{attribute 'no_assign'}
{attribute 'no_explicit_call' := 'do not call this function block directly'}
FUNCTION_BLOCK ListAppendGenericTest EXTENDS TOF_Testing.SingleCycleTest
VAR_STAT
	{attribute 'hide'}
	_ClassName : STRING := __POUNAME();
END_VAR
VAR
	_List : TOF_Collections.IList;
	_Values : ARRAY [0..5] OF STRING := ['String0', 'String1', 'String2', 'String3', 'String4', 'String5'];
END_VAR

(*!
<summary>Clears the fixture before the runner publishes the result.</summary>
<description>
Also runs after an unexpected exception interrupts the case.
</description>
*)
METHOD PROTECTED AfterTest
_List.Clear();
END_METHOD

//! <summary>Borrows the concrete class name. Callers must not modify it.</summary>
{attribute 'monitoring' := 'call'}
PROPERTY ClassName : REFERENCE TO STRING
GET
ClassName REF= _ClassName;
END_GET
END_PROPERTY

(*!
<summary>Checks appending borrowed strings without cloning or adopting them.</summary>
*)
METHOD PROTECTED ExecuteTest
VAR
	entry : TOF_Core.GENERIC_VALUE;
	expected : ARRAY [0..2] OF STRING := ['String0', 'String1', 'String2'];
	i : DINT;
END_VAR
entry := TOF_Core.GenericValueFactory.FromStringReference(value := _Values[0]);
_List.AppendGeneric(value := entry);

entry := TOF_Core.GenericValueFactory.FromStringReference(value := _Values[1]);
_List.AppendGeneric(value := entry);

entry := TOF_Core.GenericValueFactory.FromStringReference(value := _Values[2]);
_List.AppendGeneric(value := entry);

Assert.ThatBool(
	actual := _List.Get(index := 2).Address = entry.Address AND_THEN NOT _List.Get(index := 2).IsMemoryOwner,
	message := "AppendGeneric must retain the borrowed address and ownership mode"
).IsTrue();

Assert.ThatDInt(
	actual := _List.Length,
	message := "Unexpected sequence after AppendGeneric length"
).ToBe(expected := DINT#3);

FOR i := 0 TO 2 DO
	Assert.ThatString(
		actual := _List.Get(index := i).AsString255(),
		message := TOF_Core.WideStrings.Concat255("Unexpected sequence after AppendGeneric at index ", TO_WSTRING(i))
	).ToBe(expected := expected[i]);
END_FOR
END_METHOD

(*!
<summary>Binds the list fixture for this case.</summary>
<description>
Stores a borrowed interface without invoking the fixture. The owning group keeps it alive and
reserves it for this case. TestElement initializes the name and parent.
</description>
<param name="name">Display name of this case.</param>
<param name="parent">Group that owns this case.</param>
<param name="list">Required live list reserved for this case.</param>
*)
METHOD FB_init : BOOL
VAR_INPUT
	bInitRetains: BOOL; // TRUE: the retain variables are initialized (reset warm / reset cold)
	bInCopyCode: BOOL; // TRUE: the instance will be copied to the copy code afterward (online change)
	name : WSTRING;
	parent : TOF_Testing.ITestElement;
	list : TOF_Collections.IList;
END_VAR
_List := list;
FB_init := TRUE;
END_METHOD

//! <summary>Borrows the compiler-initialized namespace name. Callers must not modify it.</summary>
{attribute 'monitoring' := 'call'}
PROPERTY NamespaceName : REFERENCE TO STRING
GET
NamespaceName REF= CurrentNamespace.Name;
END_GET
END_PROPERTY

//! <summary>Reports the concrete instance size in bytes.</summary>
{attribute 'monitoring' := 'call'}
PROPERTY SelfSize : ULINT
GET
SelfSize := XSIZEOF(THIS^);
END_GET
END_PROPERTY

END_FUNCTION_BLOCK

// ---- Tests/Collections/ListInsertGenericTest.TcPOU
(*
SPDX-FileCopyrightText: c 2026 Oleksandr Tiutyk <trofimich@gmail.com>
SPDX-License-Identifier: MIT
License: https://opensource.org/license/mit
*)

(*!
<summary>Checks borrowed insertion and suffix order.</summary>
<description>
Borrows a group-owned list reserved for this case. Use from one task at a stable address.
Teardown clears the list before publication.
</description>
*)

{attribute 'no_assign'}
{attribute 'no_explicit_call' := 'do not call this function block directly'}
FUNCTION_BLOCK ListInsertGenericTest EXTENDS TOF_Testing.SingleCycleTest
VAR_STAT
	{attribute 'hide'}
	_ClassName : STRING := __POUNAME();
END_VAR
VAR
	_List : TOF_Collections.IList;
	_Values : ARRAY [0..5] OF STRING := ['String0', 'String1', 'String2', 'String3', 'String4', 'String5'];
END_VAR

(*!
<summary>Clears the fixture before the runner publishes the result.</summary>
<description>
Also runs after an unexpected exception interrupts the case.
</description>
*)
METHOD PROTECTED AfterTest
_List.Clear();
END_METHOD

//! <summary>Borrows the concrete class name. Callers must not modify it.</summary>
{attribute 'monitoring' := 'call'}
PROPERTY ClassName : REFERENCE TO STRING
GET
ClassName REF= _ClassName;
END_GET
END_PROPERTY

(*!
<summary>Checks borrowed insertion and suffix order.</summary>
*)
METHOD PROTECTED ExecuteTest
VAR
	values : ARRAY [0..5] OF STRING := ['String0', 'String1', 'String2', 'String3', 'String4', 'String5'];
	entry : TOF_Core.GENERIC_VALUE;
	expected : ARRAY [0..3] OF STRING := ['String0', 'String5', 'String1', 'String2'];
	i : DINT;
END_VAR
_List.AppendCopy(value := values[0]);
_List.AppendCopy(value := values[1]);
_List.AppendCopy(value := values[2]);

entry := TOF_Core.GenericValueFactory.FromStringReference(value := _Values[5]);
_List.InsertGeneric(index := 1, value := entry);

Assert.ThatBool(
	actual := _List.Get(index := 1).Address = entry.Address AND_THEN NOT _List.Get(index := 1).IsMemoryOwner,
	message := "InsertGeneric must retain the borrowed address and ownership mode"
).IsTrue();

Assert.ThatDInt(
	actual := _List.Length,
	message := "Unexpected sequence after InsertGeneric length"
).ToBe(expected := DINT#4);

FOR i := 0 TO 3 DO
	Assert.ThatString(
		actual := _List.Get(index := i).AsString255(),
		message := TOF_Core.WideStrings.Concat255("Unexpected sequence after InsertGeneric at index ", TO_WSTRING(i))
	).ToBe(expected := expected[i]);
END_FOR
END_METHOD

(*!
<summary>Binds the list fixture for this case.</summary>
<description>
Stores a borrowed interface without invoking the fixture. The owning group keeps it alive and
reserves it for this case. TestElement initializes the name and parent.
</description>
<param name="name">Display name of this case.</param>
<param name="parent">Group that owns this case.</param>
<param name="list">Required live list reserved for this case.</param>
*)
METHOD FB_init : BOOL
VAR_INPUT
	bInitRetains: BOOL; // TRUE: the retain variables are initialized (reset warm / reset cold)
	bInCopyCode: BOOL; // TRUE: the instance will be copied to the copy code afterward (online change)
	name : WSTRING;
	parent : TOF_Testing.ITestElement;
	list : TOF_Collections.IList;
END_VAR
_List := list;
FB_init := TRUE;
END_METHOD

//! <summary>Borrows the compiler-initialized namespace name. Callers must not modify it.</summary>
{attribute 'monitoring' := 'call'}
PROPERTY NamespaceName : REFERENCE TO STRING
GET
NamespaceName REF= CurrentNamespace.Name;
END_GET
END_PROPERTY

//! <summary>Reports the concrete instance size in bytes.</summary>
{attribute 'monitoring' := 'call'}
PROPERTY SelfSize : ULINT
GET
SelfSize := XSIZEOF(THIS^);
END_GET
END_PROPERTY

END_FUNCTION_BLOCK

// ---- Tests/Collections/ListGetAndSetGenericTest.TcPOU
(*
SPDX-FileCopyrightText: c 2026 Oleksandr Tiutyk <trofimich@gmail.com>
SPDX-License-Identifier: MIT
License: https://opensource.org/license/mit
*)

(*!
<summary>Checks borrowed replacement and the surrounding entries.</summary>
<description>
Borrows a group-owned list reserved for this case. Use from one task at a stable address.
Teardown clears the list before publication.
</description>
*)

{attribute 'no_assign'}
{attribute 'no_explicit_call' := 'do not call this function block directly'}
FUNCTION_BLOCK ListGetAndSetGenericTest EXTENDS TOF_Testing.SingleCycleTest
VAR_STAT
	{attribute 'hide'}
	_ClassName : STRING := __POUNAME();
END_VAR
VAR
	_List : TOF_Collections.IList;
	_Values : ARRAY [0..5] OF STRING := ['String0', 'String1', 'String2', 'String3', 'String4', 'String5'];
END_VAR

(*!
<summary>Clears the fixture before the runner publishes the result.</summary>
<description>
Also runs after an unexpected exception interrupts the case.
</description>
*)
METHOD PROTECTED AfterTest
_List.Clear();
END_METHOD

//! <summary>Borrows the concrete class name. Callers must not modify it.</summary>
{attribute 'monitoring' := 'call'}
PROPERTY ClassName : REFERENCE TO STRING
GET
ClassName REF= _ClassName;
END_GET
END_PROPERTY

(*!
<summary>Checks borrowed replacement and the surrounding entries.</summary>
*)
METHOD PROTECTED ExecuteTest
VAR
	values : ARRAY [0..5] OF STRING := ['String0', 'String1', 'String2', 'String3', 'String4', 'String5'];
	entry : TOF_Core.GENERIC_VALUE;
	expected : ARRAY [0..2] OF STRING := ['String0', 'String4', 'String2'];
	i : DINT;
END_VAR
_List.AppendCopy(value := values[0]);
_List.AppendCopy(value := values[1]);
_List.AppendCopy(value := values[2]);

entry := TOF_Core.GenericValueFactory.FromStringReference(value := _Values[4]);
_List.SetGeneric(index := 1, value := entry);

Assert.ThatBool(
	actual := _List.Get(index := 1).Address = entry.Address AND_THEN NOT _List.Get(index := 1).IsMemoryOwner,
	message := "SetGeneric must retain the borrowed address and ownership mode"
).IsTrue();

Assert.ThatDInt(
	actual := _List.Length,
	message := "Unexpected sequence after GetAndSetGeneric length"
).ToBe(expected := DINT#3);

FOR i := 0 TO 2 DO
	Assert.ThatString(
		actual := _List.Get(index := i).AsString255(),
		message := TOF_Core.WideStrings.Concat255("Unexpected sequence after GetAndSetGeneric at index ", TO_WSTRING(i))
	).ToBe(expected := expected[i]);
END_FOR
END_METHOD

(*!
<summary>Binds the list fixture for this case.</summary>
<description>
Stores a borrowed interface without invoking the fixture. The owning group keeps it alive and
reserves it for this case. TestElement initializes the name and parent.
</description>
<param name="name">Display name of this case.</param>
<param name="parent">Group that owns this case.</param>
<param name="list">Required live list reserved for this case.</param>
*)
METHOD FB_init : BOOL
VAR_INPUT
	bInitRetains: BOOL; // TRUE: the retain variables are initialized (reset warm / reset cold)
	bInCopyCode: BOOL; // TRUE: the instance will be copied to the copy code afterward (online change)
	name : WSTRING;
	parent : TOF_Testing.ITestElement;
	list : TOF_Collections.IList;
END_VAR
_List := list;
FB_init := TRUE;
END_METHOD

//! <summary>Borrows the compiler-initialized namespace name. Callers must not modify it.</summary>
{attribute 'monitoring' := 'call'}
PROPERTY NamespaceName : REFERENCE TO STRING
GET
NamespaceName REF= CurrentNamespace.Name;
END_GET
END_PROPERTY

//! <summary>Reports the concrete instance size in bytes.</summary>
{attribute 'monitoring' := 'call'}
PROPERTY SelfSize : ULINT
GET
SelfSize := XSIZEOF(THIS^);
END_GET
END_PROPERTY

END_FUNCTION_BLOCK

// ---- Tests/Collections/Dynamic/DynamicListClearTest.TcPOU
(*
SPDX-FileCopyrightText: c 2026 Oleksandr Tiutyk <trofimich@gmail.com>
SPDX-License-Identifier: MIT
License: https://opensource.org/license/mit
*)

(*!
<summary>Checks release of populated storage and fresh allocation on reuse.</summary>
<description>
Owns a list and its copied entries. Use from one task at a stable address.
Teardown clears surviving entries before publication.
</description>
*)

{attribute 'no_assign'}
{attribute 'no_explicit_call' := 'do not call this function block directly'}
FUNCTION_BLOCK DynamicListClearTest EXTENDS TOF_Testing.SingleCycleTest
VAR_STAT
	{attribute 'hide'}
	_ClassName : STRING := __POUNAME();
END_VAR
VAR
	_List : TOF_Collections.List<0>(valueValidator := 0);
END_VAR

(*!
<summary>Checks release of populated storage and fresh allocation on reuse.</summary>
*)
METHOD PROTECTED ExecuteTest
VAR
	values : ARRAY [0..5] OF STRING := ['String0', 'String1', 'String2', 'String3', 'String4', 'String5'];
END_VAR
_List.AppendCopy(value := values[0]);
_List.AppendCopy(value := values[1]);
_List.AppendCopy(value := values[2]);
_List.AppendCopy(value := values[3]);
_List.AppendCopy(value := values[4]);
_List.AppendCopy(value := values[5]);

Assert.ThatBool(
	actual := _List.Length = 6 AND_THEN _List.Capacity >= 6,
	message := "Clear fixture must contain six live entries"
).IsTrue();

_List.Clear();

Assert.ThatBool(
	actual := _List.Empty AND_THEN _List.Length = 0 AND_THEN _List.Capacity = 0,
	message := "Clear must empty the dynamic list and release its capacity"
).IsTrue();

_List.AppendCopy(value := values[5]);

Assert.ThatBool(
	actual := _List.Length = 1 AND_THEN _List.Get(index := 0).AsString255() = 'String5',
	message := "The cleared list must accept a fresh value"
).IsTrue();
END_METHOD

(*!
<summary>Clears the fixture before the runner publishes the result.</summary>
<description>
Also runs after an unexpected exception interrupts the case.
</description>
*)
METHOD PROTECTED AfterTest
_List.Clear();
END_METHOD

//! <summary>Borrows the concrete class name. Callers must not modify it.</summary>
{attribute 'monitoring' := 'call'}
PROPERTY ClassName : REFERENCE TO STRING
GET
ClassName REF= _ClassName;
END_GET
END_PROPERTY

//! <summary>Borrows the compiler-initialized namespace name. Callers must not modify it.</summary>
{attribute 'monitoring' := 'call'}
PROPERTY NamespaceName : REFERENCE TO STRING
GET
NamespaceName REF= CurrentNamespace.Name;
END_GET
END_PROPERTY

//! <summary>Reports the concrete instance size in bytes.</summary>
{attribute 'monitoring' := 'call'}
PROPERTY SelfSize : ULINT
GET
SelfSize := XSIZEOF(THIS^);
END_GET
END_PROPERTY

END_FUNCTION_BLOCK

// ---- Tests/Collections/Static/StaticListTestGroup.TcPOU
(*
SPDX-FileCopyrightText: c 2026 Oleksandr Tiutyk <trofimich@gmail.com>
SPDX-License-Identifier: MIT
License: https://opensource.org/license/mit
*)

(*!
<summary>Groups fixed-capacity list copying, borrowing, editing, search, sorting and overflow cases.</summary>
<description>
Owns the cases, their fixed registration array and any fixtures borrowed by the cases.
Each borrowed fixture is reserved for its case throughout the group lifetime. Use from one task at a stable address.
</description>
*)

{attribute 'no_assign'}
{attribute 'no_explicit_call' := 'do not call this function block directly'}
FUNCTION_BLOCK StaticListTestGroup EXTENDS TOF_Testing.TestGroup<16>
VAR_STAT
	{attribute 'hide'}
	_ClassName : STRING := __POUNAME();
END_VAR
VAR
	_AppendList : TOF_Collections.List<8>(valueValidator := 0);
	_InsertList : TOF_Collections.List<8>(valueValidator := 0);
	_GetAndSetList : TOF_Collections.List<8>(valueValidator := 0);
	_FindList : TOF_Collections.List<8>(valueValidator := 0);
	_ContainsList : TOF_Collections.List<8>(valueValidator := 0);
	_ContainsGenericList : TOF_Collections.List<8>(valueValidator := 0);
	_RemoveFirstList : TOF_Collections.List<8>(valueValidator := 0);
	_RemoveMatchedList : TOF_Collections.List<8>(valueValidator := 0);
	_RemoveAtList : TOF_Collections.List<8>(valueValidator := 0);
	_SwapList : TOF_Collections.List<8>(valueValidator := 0);
	_AppendGenericList : TOF_Collections.List<8>(valueValidator := 0);
	_InsertGenericList : TOF_Collections.List<8>(valueValidator := 0);
	_GetAndSetGenericList : TOF_Collections.List<8>(valueValidator := 0);

	_Append : ListAppendTest(name := "Append", parent := THIS^, list := _AppendList);
	_Insert : ListInsertTest(name := "Insert", parent := THIS^, list := _InsertList);
	_GetAndSet : ListGetAndSetTest(name := "GetAndSet", parent := THIS^, list := _GetAndSetList);
	_Find : ListFindTest(name := "Find", parent := THIS^, list := _FindList);
	_Contains : ListContainsTest(name := "Contains", parent := THIS^, list := _ContainsList);
	_ContainsGeneric : ListContainsGenericTest(name := "ContainsGeneric", parent := THIS^, list := _ContainsGenericList);
	_RemoveFirst : ListRemoveFirstTest(name := "RemoveFirst", parent := THIS^, list := _RemoveFirstList);
	_RemoveMatched : ListRemoveMatchedTest(name := "RemoveMatched", parent := THIS^, list := _RemoveMatchedList);
	_RemoveAt : ListRemoveAtTest(name := "RemoveAt", parent := THIS^, list := _RemoveAtList);
	_Swap : ListSwapTest(name := "Swap", parent := THIS^, list := _SwapList);
	_Sort : StaticListSortTest(name := "Sort", parent := THIS^);
	_AppendGeneric : ListAppendGenericTest(name := "AppendGeneric", parent := THIS^, list := _AppendGenericList);
	_InsertGeneric : ListInsertGenericTest(name := "InsertGeneric", parent := THIS^, list := _InsertGenericList);
	_GetAndSetGeneric : ListGetAndSetGenericTest(
		name := "GetAndSetGeneric",
		parent := THIS^,
		list := _GetAndSetGenericList
	);
	_Clear : StaticListClearTest(name := "Clear", parent := THIS^);
	_Overflow : StaticListOverflowTest(name := "Overflow", parent := THIS^);

	_Children : ARRAY [0.._ChildCount - 1] OF TOF_Testing.ITestElement :=
	[
		_Append,
		_Insert,
		_GetAndSet,
		_Find,
		_Contains,
		_ContainsGeneric,
		_RemoveFirst,
		_RemoveMatched,
		_RemoveAt,
		_Swap,
		_Sort,
		_AppendGeneric,
		_InsertGeneric,
		_GetAndSetGeneric,
		_Clear,
		_Overflow
	];
END_VAR

//! <summary>Borrows the fixed child array. Callers must not modify it.</summary>
{attribute 'monitoring' := 'call'}
PROPERTY Children : REFERENCE TO ARRAY [0.._ChildCount - 1] OF TOF_Testing.ITestElement
GET
Children REF= _Children;
END_GET
END_PROPERTY

//! <summary>Borrows the concrete class name. Callers must not modify it.</summary>
{attribute 'monitoring' := 'call'}
PROPERTY ClassName : REFERENCE TO STRING
GET
ClassName REF= _ClassName;
END_GET
END_PROPERTY

//! <summary>Borrows the compiler-initialized namespace name. Callers must not modify it.</summary>
{attribute 'monitoring' := 'call'}
PROPERTY NamespaceName : REFERENCE TO STRING
GET
NamespaceName REF= CurrentNamespace.Name;
END_GET
END_PROPERTY

//! <summary>Reports the concrete instance size in bytes.</summary>
{attribute 'monitoring' := 'call'}
PROPERTY SelfSize : ULINT
GET
SelfSize := XSIZEOF(THIS^);
END_GET
END_PROPERTY

END_FUNCTION_BLOCK

// ---- Tests/Collections/Static/StaticListSortTest.TcPOU
(*
SPDX-FileCopyrightText: c 2026 Oleksandr Tiutyk <trofimich@gmail.com>
SPDX-License-Identifier: MIT
License: https://opensource.org/license/mit
*)

(*!
<summary>Checks ascending sorting of a full list with duplicate strings and reverse lookup.</summary>
<description>
Owns a list and its copied entries. Use from one task at a stable address.
Teardown clears surviving entries before publication.
</description>
*)

{attribute 'no_assign'}
{attribute 'no_explicit_call' := 'do not call this function block directly'}
FUNCTION_BLOCK StaticListSortTest EXTENDS TOF_Testing.SingleCycleTest
VAR_STAT
	{attribute 'hide'}
	_ClassName : STRING := __POUNAME();
END_VAR
VAR
	_List : TOF_Collections.List<8>(valueValidator := 0);
	_Predicate : ListStringPredicate;
END_VAR

(*!
<summary>Checks ascending sorting of a full list with duplicate strings and reverse lookup.</summary>
*)
METHOD PROTECTED ExecuteTest
VAR
	values : ARRAY [0..5] OF STRING := ['String0', 'String1', 'String2', 'String3', 'String4', 'String5'];
	expected : ARRAY [0..7] OF STRING :=
		['String0', 'String1', 'String2', 'String2', 'String2', 'String3', 'String4', 'String5'];
	i : DINT;
	index : TOF_Core.DINT_INDEX;
	found : BOOL;
	entry : TOF_Core.GENERIC_VALUE;
END_VAR
_List.AppendCopy(value := values[5]);
_List.AppendCopy(value := values[4]);
_List.AppendCopy(value := values[3]);
_List.AppendCopy(value := values[2]);
_List.AppendCopy(value := values[2]);
_List.AppendCopy(value := values[2]);
_List.AppendCopy(value := values[1]);
_List.AppendCopy(value := values[0]);

_List.Sort(comparer := TOF_Comparison.StandardComparers.StringComparer);

Assert.ThatDInt(
	actual := _List.Length,
	message := "Ascending sort length"
).ToBe(expected := DINT#8);

FOR i := 0 TO 7 DO
	Assert.ThatString(
		actual := _List.Get(index := i).AsString255(),
		message := TOF_Core.WideStrings.Concat255("Ascending sort at index ", TO_WSTRING(i))
	).ToBe(expected := expected[i]);
END_FOR

_Predicate.Expected := 'String3';

found := _List.FindSingle(
	predicate := _Predicate,
	searchDirection := TOF_Core.SEARCH_DIRECTION.FROM_END,
	value => entry,
	index => index
);

Assert.ThatBool(
	actual := found AND_THEN index = 5 AND_THEN entry.AsString255() = 'String3',
	message := "Reverse lookup must return String3 at its current position after sorting"
).IsTrue();
END_METHOD

(*!
<summary>Clears the fixture before the runner publishes the result.</summary>
<description>
Also runs after an unexpected exception interrupts the case.
</description>
*)
METHOD PROTECTED AfterTest
_List.Clear();
END_METHOD

//! <summary>Borrows the concrete class name. Callers must not modify it.</summary>
{attribute 'monitoring' := 'call'}
PROPERTY ClassName : REFERENCE TO STRING
GET
ClassName REF= _ClassName;
END_GET
END_PROPERTY

//! <summary>Borrows the compiler-initialized namespace name. Callers must not modify it.</summary>
{attribute 'monitoring' := 'call'}
PROPERTY NamespaceName : REFERENCE TO STRING
GET
NamespaceName REF= CurrentNamespace.Name;
END_GET
END_PROPERTY

//! <summary>Reports the concrete instance size in bytes.</summary>
{attribute 'monitoring' := 'call'}
PROPERTY SelfSize : ULINT
GET
SelfSize := XSIZEOF(THIS^);
END_GET
END_PROPERTY

END_FUNCTION_BLOCK

// ---- Tests/Collections/Static/StaticListClearTest.TcPOU
(*
SPDX-FileCopyrightText: c 2026 Oleksandr Tiutyk <trofimich@gmail.com>
SPDX-License-Identifier: MIT
License: https://opensource.org/license/mit
*)

(*!
<summary>Checks clearing a full inline list and reusing all eight slots.</summary>
<description>
Owns a list and its copied entries. Use from one task at a stable address.
Teardown clears surviving entries before publication.
</description>
*)

{attribute 'no_assign'}
{attribute 'no_explicit_call' := 'do not call this function block directly'}
FUNCTION_BLOCK StaticListClearTest EXTENDS TOF_Testing.SingleCycleTest
VAR_STAT
	{attribute 'hide'}
	_ClassName : STRING := __POUNAME();
END_VAR
VAR
	_List : TOF_Collections.List<8>(valueValidator := 0);
END_VAR

(*!
<summary>Checks clearing a full inline list and reusing all eight slots.</summary>
*)
METHOD PROTECTED ExecuteTest
VAR
	values : ARRAY [0..5] OF STRING := ['String0', 'String1', 'String2', 'String3', 'String4', 'String5'];
END_VAR
_List.AppendCopy(value := values[0]);
_List.AppendCopy(value := values[1]);
_List.AppendCopy(value := values[2]);
_List.AppendCopy(value := values[3]);
_List.AppendCopy(value := values[4]);
_List.AppendCopy(value := values[5]);
_List.AppendCopy(value := values[0]);
_List.AppendCopy(value := values[1]);

Assert.ThatBool(
	actual := _List.Full,
	message := "Clear fixture must start full"
).IsTrue();

_List.Clear();

Assert.ThatBool(
	actual := _List.Empty AND_THEN _List.Length = 0 AND_THEN _List.Capacity = 8 AND_THEN NOT _List.Full,
	message := "Clear must empty the list while retaining its inline capacity"
).IsTrue();

_List.AppendCopy(value := values[5]);
_List.AppendCopy(value := values[4]);
_List.AppendCopy(value := values[3]);
_List.AppendCopy(value := values[2]);
_List.AppendCopy(value := values[1]);
_List.AppendCopy(value := values[0]);
_List.AppendCopy(value := values[3]);
_List.AppendCopy(value := values[4]);

Assert.ThatBool(
	actual := _List.Full AND_THEN _List.Get(index := 0).AsString255() = 'String5'
		AND_THEN _List.Get(index := 7).AsString255() = 'String4',
	message := "Refill must occupy all slots with the new head and tail"
).IsTrue();
END_METHOD

(*!
<summary>Clears the fixture before the runner publishes the result.</summary>
<description>
Also runs after an unexpected exception interrupts the case.
</description>
*)
METHOD PROTECTED AfterTest
_List.Clear();
END_METHOD

//! <summary>Borrows the concrete class name. Callers must not modify it.</summary>
{attribute 'monitoring' := 'call'}
PROPERTY ClassName : REFERENCE TO STRING
GET
ClassName REF= _ClassName;
END_GET
END_PROPERTY

//! <summary>Borrows the compiler-initialized namespace name. Callers must not modify it.</summary>
{attribute 'monitoring' := 'call'}
PROPERTY NamespaceName : REFERENCE TO STRING
GET
NamespaceName REF= CurrentNamespace.Name;
END_GET
END_PROPERTY

//! <summary>Reports the concrete instance size in bytes.</summary>
{attribute 'monitoring' := 'call'}
PROPERTY SelfSize : ULINT
GET
SelfSize := XSIZEOF(THIS^);
END_GET
END_PROPERTY

END_FUNCTION_BLOCK

// ---- Tests/Collections/Static/StaticListOverflowTest.TcPOU
(*
SPDX-FileCopyrightText: c 2026 Oleksandr Tiutyk <trofimich@gmail.com>
SPDX-License-Identifier: MIT
License: https://opensource.org/license/mit
*)

(*!
<summary>Checks overflow at eight elements and reuse after freeing a slot.</summary>
<description>
Owns a list and its copied entries. Use from one task at a stable address.
Teardown clears surviving entries before publication.
</description>
*)

{attribute 'no_assign'}
{attribute 'no_explicit_call' := 'do not call this function block directly'}
FUNCTION_BLOCK StaticListOverflowTest EXTENDS TOF_Testing.SingleCycleTest
VAR_STAT
	{attribute 'hide'}
	_ClassName : STRING := __POUNAME();
END_VAR
VAR
	_List : TOF_Collections.List<8>(valueValidator := 0);
END_VAR

(*!
<summary>Checks overflow at eight elements and reuse after freeing a slot.</summary>
*)
METHOD PROTECTED ExecuteTest
VAR
	values : ARRAY [1..9] OF INT := [1, 2, 3, 4, 5, 6, 7, 8, 9];
	i : DINT;

	exceptionCode : __SYSTEM.ExceptionCode;
	caught : TOF_Core.IException;
	fullException : TOF_Core.IStaticCollectionFullException;
END_VAR
FOR i := 1 TO 8 DO
	_List.AppendCopy(value := values[i]);
END_FOR

Assert.ThatBool(
	actual := _List.Full,
	message := "Overflow fixture must start full"
).IsTrue();

__TRY
	_List.AppendCopy(value := values[9]);
__CATCH(exceptionCode)
	caught := TOF_Core.ExceptionManager.GetLastException(
		exceptionCode := exceptionCode,
		catchPointNamespaceName := NamespaceName,
		catchPointPOUName := __POUNAME(),
		catchPointPosition := __POSITION()
	);
__ENDTRY

Assert.ThatBool(
	actual := __QUERYINTERFACE(caught, fullException),
	message := "Appending beyond capacity must raise StaticCollectionFullException"
).IsTrue();

Assert.ThatBool(
	actual := _List.Full AND_THEN _List.Length = 8 AND_THEN _List.Capacity = 8,
	message := "Rejected append must preserve length and capacity"
).IsTrue();

FOR i := 1 TO 8 DO
	Assert.ThatInt(
		actual := _List.Get(index := i - 1).AsInt(),
		message := TOF_Core.WideStrings.Concat255("Overflow must preserve member ", TO_WSTRING(i))
	).ToBe(expected := values[i]);
END_FOR

_List.RemoveAt(index := 7);
_List.AppendCopy(value := values[9]);

Assert.ThatBool(
	actual := _List.Full AND_THEN _List.Get(index := 7).AsInt() = INT#9,
	message := "Appending after removal must reuse the freed slot"
).IsTrue();
END_METHOD

(*!
<summary>Clears the fixture before the runner publishes the result.</summary>
<description>
Also runs after an unexpected exception interrupts the case.
</description>
*)
METHOD PROTECTED AfterTest
_List.Clear();
END_METHOD

//! <summary>Borrows the concrete class name. Callers must not modify it.</summary>
{attribute 'monitoring' := 'call'}
PROPERTY ClassName : REFERENCE TO STRING
GET
ClassName REF= _ClassName;
END_GET
END_PROPERTY

//! <summary>Borrows the compiler-initialized namespace name. Callers must not modify it.</summary>
{attribute 'monitoring' := 'call'}
PROPERTY NamespaceName : REFERENCE TO STRING
GET
NamespaceName REF= CurrentNamespace.Name;
END_GET
END_PROPERTY

//! <summary>Reports the concrete instance size in bytes.</summary>
{attribute 'monitoring' := 'call'}
PROPERTY SelfSize : ULINT
GET
SelfSize := XSIZEOF(THIS^);
END_GET
END_PROPERTY

END_FUNCTION_BLOCK

// ---- Tests/Collections/Dynamic/DynamicStackTestGroup.TcPOU
(*
SPDX-FileCopyrightText: c 2026 Oleksandr Tiutyk <trofimich@gmail.com>
SPDX-License-Identifier: MIT
License: https://opensource.org/license/mit
*)

(*!
<summary>Groups dynamic stack storage, LIFO order, cursors and ownership cases.</summary>
<description>
Owns the cases, their fixed registration array and any fixtures borrowed by the cases.
Each borrowed fixture is reserved for its case throughout the group lifetime. Use from one task at a stable address.
</description>
*)

{attribute 'no_assign'}
{attribute 'no_explicit_call' := 'do not call this function block directly'}
FUNCTION_BLOCK DynamicStackTestGroup EXTENDS TOF_Testing.TestGroup<11>
VAR_STAT
	{attribute 'hide'}
	_ClassName : STRING := __POUNAME();
END_VAR
VAR
	_Validator : TOF_Core.GenericValueTypeValidator(typeClass := TOF_Core.GENERIC_TYPE_CLASS.INT_16);
	_OwnedObjectCleanupStack : TOF_Collections.Stack<0>(valueValidator := 0);
	_ValidatorRejectionStack : TOF_Collections.Stack<0>(valueValidator := _Validator);
	_IndexedAccessAndEnumerationStack : TOF_Collections.Stack<0>(valueValidator := 0);
	_EmptyAndIndexBoundsStack : TOF_Collections.Stack<0>(valueValidator := 0);
	_CopiedAndBorrowedValuesStack : TOF_Collections.Stack<0>(valueValidator := 0);
	_ContainsStack : TOF_Collections.Stack<0>(valueValidator := 0);
	_ContainsGenericStack : TOF_Collections.Stack<0>(valueValidator := 0);
	_PushAndPeekStack : TOF_Collections.Stack<0>(valueValidator := 0);
	_RemoveLastStack : TOF_Collections.Stack<0>(valueValidator := 0);

	_OwnedObjectCleanup : StackOwnedObjectCleanupTest(
		name := "OwnedObjectCleanup",
		parent := THIS^,
		stack := _OwnedObjectCleanupStack
	);
	_ValidatorRejection : StackValidatorRejectionTest(
		name := "ValidatorRejection",
		parent := THIS^,
		stack := _ValidatorRejectionStack
	);
	_GrowthAndInvalidIncrement : DynamicStackGrowthAndInvalidIncrementTest(
		name := "GrowthAndInvalidIncrement",
		parent := THIS^
	);
	_IndexedAccessAndEnumeration : StackIndexedAccessAndEnumerationTest(
		name := "IndexedAccessAndEnumeration",
		parent := THIS^,
		stack := _IndexedAccessAndEnumerationStack
	);
	_EmptyAndIndexBounds : StackEmptyAndIndexBoundsTest(
		name := "EmptyAndIndexBounds",
		parent := THIS^,
		stack := _EmptyAndIndexBoundsStack
	);
	_CopiedAndBorrowedValues : StackCopiedAndBorrowedValuesTest(
		name := "CopiedAndBorrowedValues",
		parent := THIS^,
		stack := _CopiedAndBorrowedValuesStack
	);
	_Contains : StackContainsTest(name := "Contains", parent := THIS^, stack := _ContainsStack);
	_ContainsGeneric : StackContainsGenericTest(
		name := "ContainsGeneric",
		parent := THIS^,
		stack := _ContainsGenericStack
	);
	_PushAndPeek : StackPushAndPeekTest(name := "PushAndPeek", parent := THIS^, stack := _PushAndPeekStack);
	_Clear : DynamicStackClearTest(name := "Clear", parent := THIS^);
	_RemoveLast : StackRemoveLastTest(name := "RemoveLast", parent := THIS^, stack := _RemoveLastStack);

	_Children : ARRAY [0.._ChildCount - 1] OF TOF_Testing.ITestElement :=
	[
		_OwnedObjectCleanup,
		_ValidatorRejection,
		_GrowthAndInvalidIncrement,
		_IndexedAccessAndEnumeration,
		_EmptyAndIndexBounds,
		_CopiedAndBorrowedValues,
		_Contains,
		_ContainsGeneric,
		_PushAndPeek,
		_Clear,
		_RemoveLast
	];
END_VAR

//! <summary>Borrows the fixed child array. Callers must not modify it.</summary>
{attribute 'monitoring' := 'call'}
PROPERTY Children : REFERENCE TO ARRAY [0.._ChildCount - 1] OF TOF_Testing.ITestElement
GET
Children REF= _Children;
END_GET
END_PROPERTY

//! <summary>Borrows the concrete class name. Callers must not modify it.</summary>
{attribute 'monitoring' := 'call'}
PROPERTY ClassName : REFERENCE TO STRING
GET
ClassName REF= _ClassName;
END_GET
END_PROPERTY

//! <summary>Borrows the compiler-initialized namespace name. Callers must not modify it.</summary>
{attribute 'monitoring' := 'call'}
PROPERTY NamespaceName : REFERENCE TO STRING
GET
NamespaceName REF= CurrentNamespace.Name;
END_GET
END_PROPERTY

//! <summary>Reports the concrete instance size in bytes.</summary>
{attribute 'monitoring' := 'call'}
PROPERTY SelfSize : ULINT
GET
SelfSize := XSIZEOF(THIS^);
END_GET
END_PROPERTY

END_FUNCTION_BLOCK

// ---- Tests/Collections/StackOwnedObjectCleanupTest.TcPOU
(*
SPDX-FileCopyrightText: c 2026 Oleksandr Tiutyk <trofimich@gmail.com>
SPDX-License-Identifier: MIT
License: https://opensource.org/license/mit
*)

(*!
<summary>Checks ownership transfer and exactly-once disposal on removal and clear.</summary>
<description>
Borrows a group-owned stack reserved for this case. Use from one task at a stable address.
Teardown clears the stack and test-owned resources before publication.
</description>
*)

{attribute 'no_assign'}
{attribute 'no_explicit_call' := 'do not call this function block directly'}
FUNCTION_BLOCK StackOwnedObjectCleanupTest EXTENDS TOF_Testing.SingleCycleTest
VAR_STAT
	{attribute 'hide'}
	_ClassName : STRING := __POUNAME();
END_VAR
VAR
	_Stack : TOF_Collections.IStack;
	_Probe : POINTER TO ObjectExitProbe;
	_ExitCount : UDINT;
END_VAR

(*!
<summary>Binds the stack fixture for this case.</summary>
<description>
Stores a borrowed interface without invoking the fixture. The owning group keeps it alive and
reserves it for this case. TestElement initializes the name and parent.
</description>
<param name="name">Display name of this case.</param>
<param name="parent">Group that owns this case.</param>
<param name="stack">Required live stack reserved for this case.</param>
*)
METHOD FB_init : BOOL
VAR_INPUT
	bInitRetains: BOOL; // TRUE: the retain variables are initialized (reset warm / reset cold)
	bInCopyCode: BOOL; // TRUE: the instance will be copied to the copy code afterward (online change)
	name : WSTRING;
	parent : TOF_Testing.ITestElement;
	stack : TOF_Collections.IStack;
END_VAR
_Stack := stack;
FB_init := TRUE;
END_METHOD

(*!
<summary>Checks ownership transfer and exactly-once disposal on removal and clear.</summary>
*)
METHOD PROTECTED ExecuteTest
VAR
	i : DINT;
	entry : TOF_Core.GENERIC_VALUE;
END_VAR
_ExitCount := TOF_Core.UnsignedInt32.ZERO;

FOR i := 1 TO 2 DO
	_Probe := __NEW(ObjectExitProbe);

	IF _Probe = TOF_Core.Memory.NULL_ADDRESS THEN
		TOF_Core.DynamicMemoryManager.RaiseAllocationFailure();

		RETURN;
	END_IF

	_Probe^.ObserveExit(counter := _ExitCount);
	entry := TOF_Core.GenericValueFactory.FromAnyType(
		value := _Probe^,
		isObject := TRUE,
		memoryManagementBehavior := TOF_Core.GENERIC_MEMORY_MANAGEMENT_BEHAVIOR.STORE_ORIGINAL_REFERENCE_AND_OWNS_MEMORY
	);

	_Stack.PushGeneric(value := entry);
	_Probe := 0;
	entry.Reset();
END_FOR

Assert.ThatUDInt(
	actual := _ExitCount,
	message := "Insertion must keep the adopted objects alive"
).ToBe(expected := UDINT#0);

_Stack.RemoveLast();

Assert.ThatUDInt(
	actual := _ExitCount,
	message := "RemoveLast must destroy only the top object"
).ToBe(expected := UDINT#1);

_Stack.Clear();

Assert.ThatUDInt(
	actual := _ExitCount,
	message := "Clear must destroy the remaining object"
).ToBe(expected := UDINT#2);

_Stack.Clear();

Assert.ThatUDInt(
	actual := _ExitCount,
	message := "A second Clear must not destroy an object twice"
).ToBe(expected := UDINT#2);
END_METHOD

(*!
<summary>Clears the fixture before the runner publishes the result.</summary>
<description>
Also runs after an unexpected exception interrupts the case.
</description>
*)
METHOD PROTECTED AfterTest
_Stack.Clear();

IF _Probe <> TOF_Core.Memory.NULL_ADDRESS THEN
	__DELETE(_Probe);
END_IF
END_METHOD

//! <summary>Borrows the concrete class name. Callers must not modify it.</summary>
{attribute 'monitoring' := 'call'}
PROPERTY ClassName : REFERENCE TO STRING
GET
ClassName REF= _ClassName;
END_GET
END_PROPERTY

//! <summary>Borrows the compiler-initialized namespace name. Callers must not modify it.</summary>
{attribute 'monitoring' := 'call'}
PROPERTY NamespaceName : REFERENCE TO STRING
GET
NamespaceName REF= CurrentNamespace.Name;
END_GET
END_PROPERTY

//! <summary>Reports the concrete instance size in bytes.</summary>
{attribute 'monitoring' := 'call'}
PROPERTY SelfSize : ULINT
GET
SelfSize := XSIZEOF(THIS^);
END_GET
END_PROPERTY

END_FUNCTION_BLOCK

// ---- Tests/Collections/StackValidatorRejectionTest.TcPOU
(*
SPDX-FileCopyrightText: c 2026 Oleksandr Tiutyk <trofimich@gmail.com>
SPDX-License-Identifier: MIT
License: https://opensource.org/license/mit
*)

(*!
<summary>Checks rejected ownership, unchanged storage and caller disposal.</summary>
<description>
Borrows a group-owned stack reserved for this case. Use from one task at a stable address.
Teardown clears the stack and test-owned resources before publication.
</description>
*)

{attribute 'no_assign'}
{attribute 'no_explicit_call' := 'do not call this function block directly'}
FUNCTION_BLOCK StackValidatorRejectionTest EXTENDS TOF_Testing.SingleCycleTest
VAR_STAT
	{attribute 'hide'}
	_ClassName : STRING := __POUNAME();
END_VAR
VAR
	_Stack : TOF_Collections.IStack;
	_Probe : POINTER TO ObjectExitProbe;
	_ExitCount : UDINT;
END_VAR

(*!
<summary>Clears the fixture before the runner publishes the result.</summary>
<description>
Also runs after an unexpected exception interrupts the case.
</description>
*)
METHOD PROTECTED AfterTest
_Stack.Clear();

IF _Probe <> TOF_Core.Memory.NULL_ADDRESS THEN
	__DELETE(_Probe);
END_IF
END_METHOD

//! <summary>Borrows the concrete class name. Callers must not modify it.</summary>
{attribute 'monitoring' := 'call'}
PROPERTY ClassName : REFERENCE TO STRING
GET
ClassName REF= _ClassName;
END_GET
END_PROPERTY

(*!
<summary>Checks rejected ownership, unchanged storage and caller disposal.</summary>
*)
METHOD PROTECTED ExecuteTest
VAR
	entry : TOF_Core.GENERIC_VALUE;
	originalCapacity : DINT;

	exceptionCode : __SYSTEM.ExceptionCode;
	caught : TOF_Core.IException;
	typeException : TOF_Core.IIncompatibleGenericValueTypeException;
END_VAR
_ExitCount := TOF_Core.UnsignedInt32.ZERO;
originalCapacity := _Stack.Capacity;

_Probe := __NEW(ObjectExitProbe);

IF _Probe = TOF_Core.Memory.NULL_ADDRESS THEN
	TOF_Core.DynamicMemoryManager.RaiseAllocationFailure();

	RETURN;
END_IF

_Probe^.ObserveExit(counter := _ExitCount);
entry := TOF_Core.GenericValueFactory.FromAnyType(
	value := _Probe^,
	isObject := TRUE,
	memoryManagementBehavior := TOF_Core.GENERIC_MEMORY_MANAGEMENT_BEHAVIOR.STORE_ORIGINAL_REFERENCE_AND_OWNS_MEMORY
);

__TRY
	_Stack.PushGeneric(value := entry);
	_Probe := 0;
	entry.Reset();
__CATCH(exceptionCode)
	caught := TOF_Core.ExceptionManager.GetLastException(
		exceptionCode := exceptionCode,
		catchPointNamespaceName := NamespaceName,
		catchPointPOUName := __POUNAME(),
		catchPointPosition := __POSITION()
	);
__ENDTRY

Assert.ThatBool(
	actual := __QUERYINTERFACE(caught, typeException),
	message := "INT validator must reject owned OBJECT with the expected type"
).IsTrue();

Assert.ThatBool(
	actual := _Stack.Empty AND_THEN _Stack.Capacity = originalCapacity,
	message := "Rejection must precede insertion or growth"
).IsTrue();

Assert.ThatUDInt(
	actual := _ExitCount,
	message := "A rejected object must remain alive"
).ToBe(expected := UDINT#0);

IF _Probe <> TOF_Core.Memory.NULL_ADDRESS THEN
	__DELETE(_Probe);
	entry.Reset();
END_IF

Assert.ThatUDInt(
	actual := _ExitCount,
	message := "The caller must be able to destroy the rejected object once"
).ToBe(expected := UDINT#1);
END_METHOD

(*!
<summary>Binds the stack fixture for this case.</summary>
<description>
Stores a borrowed interface without invoking the fixture. The owning group keeps it alive and
reserves it for this case. TestElement initializes the name and parent.
</description>
<param name="name">Display name of this case.</param>
<param name="parent">Group that owns this case.</param>
<param name="stack">Required live stack reserved for this case.</param>
*)
METHOD FB_init : BOOL
VAR_INPUT
	bInitRetains: BOOL; // TRUE: the retain variables are initialized (reset warm / reset cold)
	bInCopyCode: BOOL; // TRUE: the instance will be copied to the copy code afterward (online change)
	name : WSTRING;
	parent : TOF_Testing.ITestElement;
	stack : TOF_Collections.IStack;
END_VAR
_Stack := stack;
FB_init := TRUE;
END_METHOD

//! <summary>Borrows the compiler-initialized namespace name. Callers must not modify it.</summary>
{attribute 'monitoring' := 'call'}
PROPERTY NamespaceName : REFERENCE TO STRING
GET
NamespaceName REF= CurrentNamespace.Name;
END_GET
END_PROPERTY

//! <summary>Reports the concrete instance size in bytes.</summary>
{attribute 'monitoring' := 'call'}
PROPERTY SelfSize : ULINT
GET
SelfSize := XSIZEOF(THIS^);
END_GET
END_PROPERTY

END_FUNCTION_BLOCK

// ---- Tests/Collections/Dynamic/DynamicStackGrowthAndInvalidIncrementTest.TcPOU
(*
SPDX-FileCopyrightText: c 2026 Oleksandr Tiutyk <trofimich@gmail.com>
SPDX-License-Identifier: MIT
License: https://opensource.org/license/mit
*)

(*!
<summary>Checks growth, rejection of a zero increment and recovery.</summary>
<description>
Owns a stack and its copied values at a stable address. Use from one task.
Teardown clears surviving entries before publication.
</description>
*)

{attribute 'no_assign'}
{attribute 'no_explicit_call' := 'do not call this function block directly'}
FUNCTION_BLOCK DynamicStackGrowthAndInvalidIncrementTest EXTENDS TOF_Testing.SingleCycleTest
VAR_STAT
	{attribute 'hide'}
	_ClassName : STRING := __POUNAME();
END_VAR
VAR
	_Stack : TOF_Collections.Stack<0>(valueValidator := 0);
END_VAR

(*!
<summary>Checks growth, rejection of a zero increment and recovery.</summary>
*)
METHOD PROTECTED ExecuteTest
VAR
	i : DINT;
	value : INT := 99;

	exceptionCode : __SYSTEM.ExceptionCode;
	caught : TOF_Core.IException;
	rangeException : TOF_Core.IArgumentOutOfRangeException;
END_VAR
_Stack.DefaultDynamicAllocationElementCount := BYTE#2;

Assert.ThatBool(
	actual := _Stack.Dynamic,
	message := "Zero static capacity must select dynamic storage"
).IsTrue();

FOR i := 1 TO 6 DO
	_Stack.PushCopy(value := i);
END_FOR

Assert.ThatBool(
	actual := _Stack.Length = 6 AND_THEN _Stack.Capacity = 6 AND_THEN NOT _Stack.Full,
	message := "Growth must retain six entries and honor the configured increment"
).IsTrue();

FOR i := 0 TO 5 DO
	Assert.ThatDInt(
		actual := _Stack.GetByIndex(index := i).AsDInt(),
		message := "Growth must preserve LIFO order"
	).ToBe(expected := 6 - i);
END_FOR

_Stack.DefaultDynamicAllocationElementCount := BYTE#0;

__TRY
	_Stack.PushCopy(value := value);
__CATCH(exceptionCode)
	caught := TOF_Core.ExceptionManager.GetLastException(
		exceptionCode := exceptionCode,
		catchPointNamespaceName := NamespaceName,
		catchPointPOUName := __POUNAME(),
		catchPointPosition := __POSITION()
	);
__ENDTRY

Assert.ThatBool(
	actual := __QUERYINTERFACE(caught, rangeException),
	message := "Zero growth must raise ArgumentOutOfRangeException"
).IsTrue();

Assert.ThatBool(
	actual := _Stack.Length = 6 AND_THEN _Stack.Capacity = 6,
	message := "Rejected growth must preserve length and capacity"
).IsTrue();

FOR i := 0 TO 5 DO
	Assert.ThatDInt(
		actual := _Stack.GetByIndex(index := i).AsDInt(),
		message := "Rejected growth must preserve every entry"
	).ToBe(expected := 6 - i);
END_FOR

_Stack.DefaultDynamicAllocationElementCount := BYTE#2;
_Stack.PushCopy(value := value);

Assert.ThatDInt(
	actual := _Stack.Capacity,
	message := "A valid increment must allow growth after rejection"
).ToBe(expected := DINT#8);

Assert.ThatInt(
	actual := _Stack.Peek().AsInt(),
	message := "Push after rejection must establish the new top"
).ToBe(expected := value);
END_METHOD

(*!
<summary>Clears the fixture before the runner publishes the result.</summary>
<description>
Also runs after an unexpected exception interrupts the case.
</description>
*)
METHOD PROTECTED AfterTest
_Stack.Clear();
END_METHOD

//! <summary>Borrows the concrete class name. Callers must not modify it.</summary>
{attribute 'monitoring' := 'call'}
PROPERTY ClassName : REFERENCE TO STRING
GET
ClassName REF= _ClassName;
END_GET
END_PROPERTY

//! <summary>Borrows the compiler-initialized namespace name. Callers must not modify it.</summary>
{attribute 'monitoring' := 'call'}
PROPERTY NamespaceName : REFERENCE TO STRING
GET
NamespaceName REF= CurrentNamespace.Name;
END_GET
END_PROPERTY

//! <summary>Reports the concrete instance size in bytes.</summary>
{attribute 'monitoring' := 'call'}
PROPERTY SelfSize : ULINT
GET
SelfSize := XSIZEOF(THIS^);
END_GET
END_PROPERTY

END_FUNCTION_BLOCK

// ---- Tests/Collections/StackIndexedAccessAndEnumerationTest.TcPOU
(*
SPDX-FileCopyrightText: c 2026 Oleksandr Tiutyk <trofimich@gmail.com>
SPDX-License-Identifier: MIT
License: https://opensource.org/license/mit
*)

(*!
<summary>Checks top-first lookup, independent traversal, exhaustion and reset.</summary>
<description>
Borrows a group-owned stack reserved for this case. Use from one task at a stable address.
Teardown clears the stack and test-owned resources before publication.
</description>
*)

{attribute 'no_assign'}
{attribute 'no_explicit_call' := 'do not call this function block directly'}
FUNCTION_BLOCK StackIndexedAccessAndEnumerationTest EXTENDS TOF_Testing.SingleCycleTest
VAR_STAT
	{attribute 'hide'}
	_ClassName : STRING := __POUNAME();
END_VAR
VAR
	_Stack : TOF_Collections.IStack;
	_Enumerator : TOF_Core.IEnumerator;
	_SecondEnumerator : TOF_Core.IEnumerator;
END_VAR

(*!
<summary>Clears the fixture before the runner publishes the result.</summary>
<description>
Also runs after an unexpected exception interrupts the case.
</description>
*)
METHOD PROTECTED AfterTest
releaseCursor(cursor := _Enumerator);
releaseCursor(cursor := _SecondEnumerator);
_Stack.Clear();
END_METHOD

//! <summary>Borrows the concrete class name. Callers must not modify it.</summary>
{attribute 'monitoring' := 'call'}
PROPERTY ClassName : REFERENCE TO STRING
GET
ClassName REF= _ClassName;
END_GET
END_PROPERTY

(*!
<summary>Checks top-first lookup, independent traversal, exhaustion and reset.</summary>
*)
METHOD PROTECTED ExecuteTest
VAR
	values : ARRAY [1..4] OF INT := [11, 22, 33, 44];
	i : DINT;
	moved : BOOL;
END_VAR
_Stack.PushCopy(value := values[1]);
_Stack.PushCopy(value := values[2]);
_Stack.PushCopy(value := values[3]);

FOR i := 0 TO 2 DO
	Assert.ThatInt(
		actual := _Stack.GetByIndex(index := i).AsInt(),
		message := "Indexed access must run from top to bottom"
	).ToBe(expected := values[3 - i]);
END_FOR

_Enumerator := _Stack.CreateEnumerator();
_SecondEnumerator := _Stack.CreateEnumerator();

IF _Enumerator = 0 OR_ELSE _SecondEnumerator = 0 THEN
	RecordFailure(message := "Stack must create both cursors");

	RETURN;
END_IF

IF _Enumerator = _SecondEnumerator THEN
	_SecondEnumerator := 0;
	RecordFailure(message := "Two traversals must own distinct cursors");

	RETURN;
END_IF

Assert.ThatBool(
	actual := _Enumerator.Current.TypeClass = TOF_Core.GENERIC_TYPE_CLASS.UNSPECIFIED,
	message := "Current before traversal must be empty"
).IsTrue();

FOR i := 3 TO 1 BY -1 DO
	moved := _Enumerator.MoveNext();

	Assert.ThatBool(
		actual := moved AND_THEN _Enumerator.Current.AsInt() = values[i],
		message := "Cursor must visit entries in LIFO order"
	).IsTrue();
END_FOR

Assert.ThatBool(
	actual := _Enumerator.MoveNext(),
	message := "Cursor must stop at end"
).IsFalse();

Assert.ThatBool(
	actual := _Enumerator.MoveNext(),
	message := "Exhaustion must persist"
).IsFalse();

Assert.ThatBool(
	actual := _Enumerator.Current.TypeClass = TOF_Core.GENERIC_TYPE_CLASS.UNSPECIFIED,
	message := "Exhausted Current must be empty"
).IsTrue();

moved := _SecondEnumerator.MoveNext();

Assert.ThatBool(
	actual := moved AND_THEN _SecondEnumerator.Current.AsInt() = values[3],
	message := "The independent cursor must start at the top"
).IsTrue();

_Enumerator.Reset();

Assert.ThatBool(
	actual := _Enumerator.Current.TypeClass = TOF_Core.GENERIC_TYPE_CLASS.UNSPECIFIED,
	message := "Reset must clear Current"
).IsTrue();

moved := _Enumerator.MoveNext();

Assert.ThatBool(
	actual := moved AND_THEN _Enumerator.Current.AsInt() = values[3],
	message := "Reset must restart at the top"
).IsTrue();

releaseCursor(cursor := _Enumerator);
releaseCursor(cursor := _SecondEnumerator);

_Stack.Clear();
_Enumerator := _Stack.CreateEnumerator();

IF _Enumerator = 0 THEN
	RecordFailure(message := "Empty stack must create a cursor");

	RETURN;
END_IF

Assert.ThatBool(
	actual := _Enumerator.MoveNext(),
	message := "An empty cursor must have no next entry"
).IsFalse();

Assert.ThatBool(
	actual := _Enumerator.MoveNext(),
	message := "An empty cursor must stay exhausted"
).IsFalse();

Assert.ThatBool(
	actual := _Enumerator.Current.TypeClass = TOF_Core.GENERIC_TYPE_CLASS.UNSPECIFIED,
	message := "Empty Current must be unspecified"
).IsTrue();
END_METHOD

(*!
<summary>Binds the stack fixture for this case.</summary>
<description>
Stores a borrowed interface without invoking the fixture. The owning group keeps it alive and
reserves it for this case. TestElement initializes the name and parent.
</description>
<param name="name">Display name of this case.</param>
<param name="parent">Group that owns this case.</param>
<param name="stack">Required live stack reserved for this case.</param>
*)
METHOD FB_init : BOOL
VAR_INPUT
	bInitRetains: BOOL; // TRUE: the retain variables are initialized (reset warm / reset cold)
	bInCopyCode: BOOL; // TRUE: the instance will be copied to the copy code afterward (online change)
	name : WSTRING;
	parent : TOF_Testing.ITestElement;
	stack : TOF_Collections.IStack;
END_VAR
_Stack := stack;
FB_init := TRUE;
END_METHOD

//! <summary>Borrows the compiler-initialized namespace name. Callers must not modify it.</summary>
{attribute 'monitoring' := 'call'}
PROPERTY NamespaceName : REFERENCE TO STRING
GET
NamespaceName REF= CurrentNamespace.Name;
END_GET
END_PROPERTY

(*!
<summary>Releases an owned cursor and invalidates the caller handle.</summary>
<description>
Reports failed disposal without replacing an earlier test failure. Call before mutating the source stack.
</description>
<param name="cursor">Owned cursor or zero. The caller handle is cleared before attempting disposal.</param>
*)
METHOD PRIVATE releaseCursor
VAR_IN_OUT
	cursor : TOF_Core.IEnumerator;
END_VAR
VAR
	owned : TOF_Core.IObject;
END_VAR
IF cursor = 0 THEN
	RETURN;
END_IF

owned := cursor;
cursor := 0;

IF NOT TOF_Core.Memory.TryReleaseDynamicObject(instance := owned) THEN
	RecordFailure(message := "Could not release the stack cursor");
END_IF
END_METHOD

//! <summary>Reports the concrete instance size in bytes.</summary>
{attribute 'monitoring' := 'call'}
PROPERTY SelfSize : ULINT
GET
SelfSize := XSIZEOF(THIS^);
END_GET
END_PROPERTY

END_FUNCTION_BLOCK

// ---- Tests/Collections/StackEmptyAndIndexBoundsTest.TcPOU
(*
SPDX-FileCopyrightText: c 2026 Oleksandr Tiutyk <trofimich@gmail.com>
SPDX-License-Identifier: MIT
License: https://opensource.org/license/mit
*)

(*!
<summary>Checks empty operations and negative and end index rejection.</summary>
<description>
Borrows a group-owned stack reserved for this case. Use from one task at a stable address.
Teardown clears the stack and test-owned resources before publication.
</description>
*)

{attribute 'no_assign'}
{attribute 'no_explicit_call' := 'do not call this function block directly'}
FUNCTION_BLOCK StackEmptyAndIndexBoundsTest EXTENDS TOF_Testing.SingleCycleTest
VAR_STAT
	{attribute 'hide'}
	_ClassName : STRING := __POUNAME();
END_VAR
VAR
	_Stack : TOF_Collections.IStack;
END_VAR

(*!
<summary>Clears the fixture before the runner publishes the result.</summary>
<description>
Also runs after an unexpected exception interrupts the case.
</description>
*)
METHOD PROTECTED AfterTest
_Stack.Clear();
END_METHOD

//! <summary>Borrows the concrete class name. Callers must not modify it.</summary>
{attribute 'monitoring' := 'call'}
PROPERTY ClassName : REFERENCE TO STRING
GET
ClassName REF= _ClassName;
END_GET
END_PROPERTY

(*!
<summary>Checks empty operations and negative and end index rejection.</summary>
*)
METHOD PROTECTED ExecuteTest
VAR
	value : INT := 7;
	invalidIndex : DINT;
	ignoredEntry : REFERENCE TO TOF_Core.GENERIC_VALUE;

	exceptionCode : __SYSTEM.ExceptionCode;
	caught : TOF_Core.IException;
	emptyException : TOF_Core.ICollectionEmptyException;
	indexException : TOF_Core.IArgumentOutOfRangeException;
END_VAR
__TRY
	ignoredEntry REF= _Stack.Peek();
__CATCH(exceptionCode)
	caught := TOF_Core.ExceptionManager.GetLastException(
		exceptionCode := exceptionCode,
		catchPointNamespaceName := NamespaceName,
		catchPointPOUName := __POUNAME(),
		catchPointPosition := __POSITION()
	);
__ENDTRY

Assert.ThatBool(
	actual := __QUERYINTERFACE(caught, emptyException),
	message := "Peek on an empty stack must raise CollectionEmptyException"
).IsTrue();

caught := 0;

__TRY
	_Stack.RemoveLast();
__CATCH(exceptionCode)
	caught := TOF_Core.ExceptionManager.GetLastException(
		exceptionCode := exceptionCode,
		catchPointNamespaceName := NamespaceName,
		catchPointPOUName := __POUNAME(),
		catchPointPosition := __POSITION()
	);
__ENDTRY

Assert.ThatBool(
	actual := __QUERYINTERFACE(caught, emptyException),
	message := "RemoveLast on an empty stack must raise CollectionEmptyException"
).IsTrue();

Assert.ThatBool(
	actual := _Stack.Empty,
	message := "Rejected empty operations must preserve the empty stack"
).IsTrue();

_Stack.PushCopy(value := value);

// Supply an invalid runtime value to the DINT_INDEX parameter.
invalidIndex := -1;
caught := 0;

__TRY
	ignoredEntry REF= _Stack.GetByIndex(index := invalidIndex);
__CATCH(exceptionCode)
	caught := TOF_Core.ExceptionManager.GetLastException(
		exceptionCode := exceptionCode,
		catchPointNamespaceName := NamespaceName,
		catchPointPOUName := __POUNAME(),
		catchPointPosition := __POSITION()
	);
__ENDTRY

Assert.ThatBool(
	actual := __QUERYINTERFACE(caught, indexException),
	message := "Index -1 must raise ArgumentOutOfRangeException"
).IsTrue();

invalidIndex := _Stack.Length;
caught := 0;

__TRY
	ignoredEntry REF= _Stack.GetByIndex(index := invalidIndex);
__CATCH(exceptionCode)
	caught := TOF_Core.ExceptionManager.GetLastException(
		exceptionCode := exceptionCode,
		catchPointNamespaceName := NamespaceName,
		catchPointPOUName := __POUNAME(),
		catchPointPosition := __POSITION()
	);
__ENDTRY

Assert.ThatBool(
	actual := __QUERYINTERFACE(caught, indexException),
	message := "Index equal to Length must raise ArgumentOutOfRangeException"
).IsTrue();

Assert.ThatDInt(
	actual := _Stack.Length,
	message := "Rejected accesses must preserve the entry count"
).ToBe(expected := DINT#1);

Assert.ThatInt(
	actual := _Stack.Peek().AsInt(),
	message := "Rejected accesses must preserve the top"
).ToBe(expected := value);
END_METHOD

(*!
<summary>Binds the stack fixture for this case.</summary>
<description>
Stores a borrowed interface without invoking the fixture. The owning group keeps it alive and
reserves it for this case. TestElement initializes the name and parent.
</description>
<param name="name">Display name of this case.</param>
<param name="parent">Group that owns this case.</param>
<param name="stack">Required live stack reserved for this case.</param>
*)
METHOD FB_init : BOOL
VAR_INPUT
	bInitRetains: BOOL; // TRUE: the retain variables are initialized (reset warm / reset cold)
	bInCopyCode: BOOL; // TRUE: the instance will be copied to the copy code afterward (online change)
	name : WSTRING;
	parent : TOF_Testing.ITestElement;
	stack : TOF_Collections.IStack;
END_VAR
_Stack := stack;
FB_init := TRUE;
END_METHOD

//! <summary>Borrows the compiler-initialized namespace name. Callers must not modify it.</summary>
{attribute 'monitoring' := 'call'}
PROPERTY NamespaceName : REFERENCE TO STRING
GET
NamespaceName REF= CurrentNamespace.Name;
END_GET
END_PROPERTY

//! <summary>Reports the concrete instance size in bytes.</summary>
{attribute 'monitoring' := 'call'}
PROPERTY SelfSize : ULINT
GET
SelfSize := XSIZEOF(THIS^);
END_GET
END_PROPERTY

END_FUNCTION_BLOCK

// ---- Tests/Collections/StackCopiedAndBorrowedValuesTest.TcPOU
(*
SPDX-FileCopyrightText: c 2026 Oleksandr Tiutyk <trofimich@gmail.com>
SPDX-License-Identifier: MIT
License: https://opensource.org/license/mit
*)

(*!
<summary>Checks copy isolation and the lifetime of a borrowed entry.</summary>
<description>
Borrows a group-owned stack reserved for this case. Use from one task at a stable address.
Teardown clears the stack and test-owned resources before publication.
</description>
*)

{attribute 'no_assign'}
{attribute 'no_explicit_call' := 'do not call this function block directly'}
FUNCTION_BLOCK StackCopiedAndBorrowedValuesTest EXTENDS TOF_Testing.SingleCycleTest
VAR_STAT
	{attribute 'hide'}
	_ClassName : STRING := __POUNAME();
END_VAR
VAR
	_Stack : TOF_Collections.IStack;
	_SourceValue : INT;
END_VAR

(*!
<summary>Clears the fixture before the runner publishes the result.</summary>
<description>
Also runs after an unexpected exception interrupts the case.
</description>
*)
METHOD PROTECTED AfterTest
_Stack.Clear();
END_METHOD

//! <summary>Borrows the concrete class name. Callers must not modify it.</summary>
{attribute 'monitoring' := 'call'}
PROPERTY ClassName : REFERENCE TO STRING
GET
ClassName REF= _ClassName;
END_GET
END_PROPERTY

(*!
<summary>Checks copy isolation and the lifetime of a borrowed entry.</summary>
*)
METHOD PROTECTED ExecuteTest
VAR
	query : TOF_Core.GENERIC_VALUE;
END_VAR
_SourceValue := 7;
_Stack.PushCopy(value := _SourceValue);
_SourceValue := 9;

Assert.ThatInt(
	actual := _Stack.Peek().AsInt(),
	message := "PushCopy must isolate the value from later source writes"
).ToBe(expected := INT#7);

query := TOF_Core.GenericValueFactory.FromIntReference(value := _SourceValue);
_Stack.PushGeneric(value := query);
_SourceValue := 11;

Assert.ThatInt(
	actual := _Stack.Peek().AsInt(),
	message := "PushGeneric must observe the current value in borrowed storage"
).ToBe(expected := INT#11);

Assert.ThatBool(
	actual := NOT _Stack.Peek().IsMemoryOwner AND_THEN _Stack.Peek().Address = query.Address,
	message := "The stored descriptor must retain the borrowed address and ownership mode"
).IsTrue();

Assert.ThatBool(
	actual := _Stack.ContainsGeneric(value := query, releaseValue := FALSE),
	message := "Borrowed lookup must find the top"
).IsTrue();

_Stack.RemoveLast();

Assert.ThatInt(
	actual := _SourceValue,
	message := "Removing a borrowed entry must preserve its source"
).ToBe(expected := INT#11);

Assert.ThatInt(
	actual := _Stack.Peek().AsInt(),
	message := "Removing the borrowed entry must reveal the copy"
).ToBe(expected := INT#7);
END_METHOD

(*!
<summary>Binds the stack fixture for this case.</summary>
<description>
Stores a borrowed interface without invoking the fixture. The owning group keeps it alive and
reserves it for this case. TestElement initializes the name and parent.
</description>
<param name="name">Display name of this case.</param>
<param name="parent">Group that owns this case.</param>
<param name="stack">Required live stack reserved for this case.</param>
*)
METHOD FB_init : BOOL
VAR_INPUT
	bInitRetains: BOOL; // TRUE: the retain variables are initialized (reset warm / reset cold)
	bInCopyCode: BOOL; // TRUE: the instance will be copied to the copy code afterward (online change)
	name : WSTRING;
	parent : TOF_Testing.ITestElement;
	stack : TOF_Collections.IStack;
END_VAR
_Stack := stack;
FB_init := TRUE;
END_METHOD

//! <summary>Borrows the compiler-initialized namespace name. Callers must not modify it.</summary>
{attribute 'monitoring' := 'call'}
PROPERTY NamespaceName : REFERENCE TO STRING
GET
NamespaceName REF= CurrentNamespace.Name;
END_GET
END_PROPERTY

//! <summary>Reports the concrete instance size in bytes.</summary>
{attribute 'monitoring' := 'call'}
PROPERTY SelfSize : ULINT
GET
SelfSize := XSIZEOF(THIS^);
END_GET
END_PROPERTY

END_FUNCTION_BLOCK

// ---- Tests/Collections/StackContainsTest.TcPOU
(*
SPDX-FileCopyrightText: c 2026 Oleksandr Tiutyk <trofimich@gmail.com>
SPDX-License-Identifier: MIT
License: https://opensource.org/license/mit
*)

(*!
<summary>Checks raw membership without changing LIFO order.</summary>
<description>
Borrows a group-owned stack reserved for this case. Use from one task at a stable address.
Teardown clears the stack and test-owned resources before publication.
</description>
*)

{attribute 'no_assign'}
{attribute 'no_explicit_call' := 'do not call this function block directly'}
FUNCTION_BLOCK StackContainsTest EXTENDS TOF_Testing.SingleCycleTest
VAR_STAT
	{attribute 'hide'}
	_ClassName : STRING := __POUNAME();
END_VAR
VAR
	_Stack : TOF_Collections.IStack;
END_VAR

(*!
<summary>Clears the fixture before the runner publishes the result.</summary>
<description>
Also runs after an unexpected exception interrupts the case.
</description>
*)
METHOD PROTECTED AfterTest
_Stack.Clear();
END_METHOD

//! <summary>Borrows the concrete class name. Callers must not modify it.</summary>
{attribute 'monitoring' := 'call'}
PROPERTY ClassName : REFERENCE TO STRING
GET
ClassName REF= _ClassName;
END_GET
END_PROPERTY

(*!
<summary>Checks raw membership without changing LIFO order.</summary>
*)
METHOD PROTECTED ExecuteTest
VAR
	values : ARRAY [1..4] OF INT := [11, 22, 33, 44];
END_VAR
Assert.ThatBool(
	actual := _Stack.Contains(value := values[1]),
	message := "An empty stack must report absence"
).IsFalse();

_Stack.PushCopy(value := values[1]);
_Stack.PushCopy(value := values[2]);
_Stack.PushCopy(value := values[3]);

Assert.ThatBool(
	actual := _Stack.Contains(value := values[1]),
	message := "Contains must find the bottom value"
).IsTrue();

Assert.ThatBool(
	actual := _Stack.Contains(value := values[3]),
	message := "Contains must find the top value"
).IsTrue();

Assert.ThatBool(
	actual := _Stack.Contains(value := values[4]),
	message := "Contains must reject an absent value"
).IsFalse();

Assert.ThatDInt(
	actual := _Stack.Length,
	message := "Lookup must preserve all three entries"
).ToBe(expected := DINT#3);
END_METHOD

(*!
<summary>Binds the stack fixture for this case.</summary>
<description>
Stores a borrowed interface without invoking the fixture. The owning group keeps it alive and
reserves it for this case. TestElement initializes the name and parent.
</description>
<param name="name">Display name of this case.</param>
<param name="parent">Group that owns this case.</param>
<param name="stack">Required live stack reserved for this case.</param>
*)
METHOD FB_init : BOOL
VAR_INPUT
	bInitRetains: BOOL; // TRUE: the retain variables are initialized (reset warm / reset cold)
	bInCopyCode: BOOL; // TRUE: the instance will be copied to the copy code afterward (online change)
	name : WSTRING;
	parent : TOF_Testing.ITestElement;
	stack : TOF_Collections.IStack;
END_VAR
_Stack := stack;
FB_init := TRUE;
END_METHOD

//! <summary>Borrows the compiler-initialized namespace name. Callers must not modify it.</summary>
{attribute 'monitoring' := 'call'}
PROPERTY NamespaceName : REFERENCE TO STRING
GET
NamespaceName REF= CurrentNamespace.Name;
END_GET
END_PROPERTY

//! <summary>Reports the concrete instance size in bytes.</summary>
{attribute 'monitoring' := 'call'}
PROPERTY SelfSize : ULINT
GET
SelfSize := XSIZEOF(THIS^);
END_GET
END_PROPERTY

END_FUNCTION_BLOCK

// ---- Tests/Collections/StackContainsGenericTest.TcPOU
(*
SPDX-FileCopyrightText: c 2026 Oleksandr Tiutyk <trofimich@gmail.com>
SPDX-License-Identifier: MIT
License: https://opensource.org/license/mit
*)

(*!
<summary>Checks generic membership with independent borrowed queries.</summary>
<description>
Borrows a group-owned stack reserved for this case. Use from one task at a stable address.
Teardown clears the stack and test-owned resources before publication.
</description>
*)

{attribute 'no_assign'}
{attribute 'no_explicit_call' := 'do not call this function block directly'}
FUNCTION_BLOCK StackContainsGenericTest EXTENDS TOF_Testing.SingleCycleTest
VAR_STAT
	{attribute 'hide'}
	_ClassName : STRING := __POUNAME();
END_VAR
VAR
	_Stack : TOF_Collections.IStack;
END_VAR

(*!
<summary>Clears the fixture before the runner publishes the result.</summary>
<description>
Also runs after an unexpected exception interrupts the case.
</description>
*)
METHOD PROTECTED AfterTest
_Stack.Clear();
END_METHOD

//! <summary>Borrows the concrete class name. Callers must not modify it.</summary>
{attribute 'monitoring' := 'call'}
PROPERTY ClassName : REFERENCE TO STRING
GET
ClassName REF= _ClassName;
END_GET
END_PROPERTY

(*!
<summary>Checks generic membership with independent borrowed queries.</summary>
*)
METHOD PROTECTED ExecuteTest
VAR
	values : ARRAY [1..4] OF INT := [11, 22, 33, 44];
	query : TOF_Core.GENERIC_VALUE;
END_VAR
_Stack.PushCopy(value := values[1]);
_Stack.PushCopy(value := values[2]);
_Stack.PushCopy(value := values[3]);

query := TOF_Core.GenericValueFactory.FromIntReference(value := values[1]);
Assert.ThatBool(
	actual := _Stack.ContainsGeneric(value := query, releaseValue := FALSE),
	message := "Generic lookup must find the bottom value"
).IsTrue();

query := TOF_Core.GenericValueFactory.FromIntReference(value := values[3]);
Assert.ThatBool(
	actual := _Stack.ContainsGeneric(value := query, releaseValue := FALSE),
	message := "Generic lookup must find the top value"
).IsTrue();

query := TOF_Core.GenericValueFactory.FromIntReference(value := values[4]);
Assert.ThatBool(
	actual := _Stack.ContainsGeneric(value := query, releaseValue := FALSE),
	message := "Generic lookup must reject an absent value"
).IsFalse();

Assert.ThatDInt(
	actual := _Stack.Length,
	message := "Generic lookup must preserve all three entries"
).ToBe(expected := DINT#3);
END_METHOD

(*!
<summary>Binds the stack fixture for this case.</summary>
<description>
Stores a borrowed interface without invoking the fixture. The owning group keeps it alive and
reserves it for this case. TestElement initializes the name and parent.
</description>
<param name="name">Display name of this case.</param>
<param name="parent">Group that owns this case.</param>
<param name="stack">Required live stack reserved for this case.</param>
*)
METHOD FB_init : BOOL
VAR_INPUT
	bInitRetains: BOOL; // TRUE: the retain variables are initialized (reset warm / reset cold)
	bInCopyCode: BOOL; // TRUE: the instance will be copied to the copy code afterward (online change)
	name : WSTRING;
	parent : TOF_Testing.ITestElement;
	stack : TOF_Collections.IStack;
END_VAR
_Stack := stack;
FB_init := TRUE;
END_METHOD

//! <summary>Borrows the compiler-initialized namespace name. Callers must not modify it.</summary>
{attribute 'monitoring' := 'call'}
PROPERTY NamespaceName : REFERENCE TO STRING
GET
NamespaceName REF= CurrentNamespace.Name;
END_GET
END_PROPERTY

//! <summary>Reports the concrete instance size in bytes.</summary>
{attribute 'monitoring' := 'call'}
PROPERTY SelfSize : ULINT
GET
SelfSize := XSIZEOF(THIS^);
END_GET
END_PROPERTY

END_FUNCTION_BLOCK

// ---- Tests/Collections/StackPushAndPeekTest.TcPOU
(*
SPDX-FileCopyrightText: c 2026 Oleksandr Tiutyk <trofimich@gmail.com>
SPDX-License-Identifier: MIT
License: https://opensource.org/license/mit
*)

(*!
<summary>Checks the current LIFO top and length after each push.</summary>
<description>
Borrows a group-owned stack reserved for this case. Use from one task at a stable address.
Teardown clears the stack and test-owned resources before publication.
</description>
*)

{attribute 'no_assign'}
{attribute 'no_explicit_call' := 'do not call this function block directly'}
FUNCTION_BLOCK StackPushAndPeekTest EXTENDS TOF_Testing.SingleCycleTest
VAR_STAT
	{attribute 'hide'}
	_ClassName : STRING := __POUNAME();
END_VAR
VAR
	_Stack : TOF_Collections.IStack;
END_VAR

(*!
<summary>Clears the fixture before the runner publishes the result.</summary>
<description>
Also runs after an unexpected exception interrupts the case.
</description>
*)
METHOD PROTECTED AfterTest
_Stack.Clear();
END_METHOD

//! <summary>Borrows the concrete class name. Callers must not modify it.</summary>
{attribute 'monitoring' := 'call'}
PROPERTY ClassName : REFERENCE TO STRING
GET
ClassName REF= _ClassName;
END_GET
END_PROPERTY

(*!
<summary>Checks the current LIFO top and length after each push.</summary>
*)
METHOD PROTECTED ExecuteTest
VAR
	values : ARRAY [1..4] OF INT := [11, 22, 33, 44];
END_VAR
_Stack.PushCopy(value := values[1]);

Assert.ThatInt(
	actual := _Stack.Peek().AsInt(),
	message := "Push 1 must establish the new top"
).ToBe(expected := values[1]);

Assert.ThatDInt(
	actual := _Stack.Length,
	message := "Peeking after push 1 must preserve length"
).ToBe(expected := DINT#1);

_Stack.PushCopy(value := values[2]);

Assert.ThatInt(
	actual := _Stack.Peek().AsInt(),
	message := "Push 2 must establish the new top"
).ToBe(expected := values[2]);

Assert.ThatDInt(
	actual := _Stack.Length,
	message := "Peeking after push 2 must preserve length"
).ToBe(expected := DINT#2);

_Stack.PushCopy(value := values[3]);

Assert.ThatInt(
	actual := _Stack.Peek().AsInt(),
	message := "Push 3 must establish the new top"
).ToBe(expected := values[3]);

Assert.ThatDInt(
	actual := _Stack.Length,
	message := "Peeking after push 3 must preserve length"
).ToBe(expected := DINT#3);
END_METHOD

(*!
<summary>Binds the stack fixture for this case.</summary>
<description>
Stores a borrowed interface without invoking the fixture. The owning group keeps it alive and
reserves it for this case. TestElement initializes the name and parent.
</description>
<param name="name">Display name of this case.</param>
<param name="parent">Group that owns this case.</param>
<param name="stack">Required live stack reserved for this case.</param>
*)
METHOD FB_init : BOOL
VAR_INPUT
	bInitRetains: BOOL; // TRUE: the retain variables are initialized (reset warm / reset cold)
	bInCopyCode: BOOL; // TRUE: the instance will be copied to the copy code afterward (online change)
	name : WSTRING;
	parent : TOF_Testing.ITestElement;
	stack : TOF_Collections.IStack;
END_VAR
_Stack := stack;
FB_init := TRUE;
END_METHOD

//! <summary>Borrows the compiler-initialized namespace name. Callers must not modify it.</summary>
{attribute 'monitoring' := 'call'}
PROPERTY NamespaceName : REFERENCE TO STRING
GET
NamespaceName REF= CurrentNamespace.Name;
END_GET
END_PROPERTY

//! <summary>Reports the concrete instance size in bytes.</summary>
{attribute 'monitoring' := 'call'}
PROPERTY SelfSize : ULINT
GET
SelfSize := XSIZEOF(THIS^);
END_GET
END_PROPERTY

END_FUNCTION_BLOCK

// ---- Tests/Collections/Dynamic/DynamicStackClearTest.TcPOU
(*
SPDX-FileCopyrightText: c 2026 Oleksandr Tiutyk <trofimich@gmail.com>
SPDX-License-Identifier: MIT
License: https://opensource.org/license/mit
*)

(*!
<summary>Checks populated clear, storage policy and reuse.</summary>
<description>
Owns a stack and its copied values at a stable address. Use from one task.
Teardown clears surviving entries before publication.
</description>
*)

{attribute 'no_assign'}
{attribute 'no_explicit_call' := 'do not call this function block directly'}
FUNCTION_BLOCK DynamicStackClearTest EXTENDS TOF_Testing.SingleCycleTest
VAR_STAT
	{attribute 'hide'}
	_ClassName : STRING := __POUNAME();
END_VAR
VAR
	_Stack : TOF_Collections.Stack<0>(valueValidator := 0);
END_VAR

(*!
<summary>Checks populated clear, storage policy and reuse.</summary>
*)
METHOD PROTECTED ExecuteTest
VAR
	values : ARRAY [1..4] OF INT := [11, 22, 33, 44];
END_VAR
_Stack.PushCopy(value := values[1]);
_Stack.PushCopy(value := values[2]);
_Stack.PushCopy(value := values[3]);

Assert.ThatDInt(
	actual := _Stack.Length,
	message := "Clear fixture must start with three entries"
).ToBe(expected := DINT#3);

_Stack.Clear();

Assert.ThatBool(
	actual := _Stack.Empty AND_THEN _Stack.Length = 0,
	message := "Clear must empty the stack"
).IsTrue();

Assert.ThatDInt(
	actual := _Stack.Capacity,
	message := "Clear must restore the expected storage capacity"
).ToBe(expected := DINT#0);

_Stack.Clear();
_Stack.PushCopy(value := values[4]);

Assert.ThatInt(
	actual := _Stack.Peek().AsInt(),
	message := "The cleared stack must expose the fresh top"
).ToBe(expected := values[4]);

Assert.ThatDInt(
	actual := _Stack.Length,
	message := "Reuse must leave only one entry"
).ToBe(expected := DINT#1);
END_METHOD

(*!
<summary>Clears the fixture before the runner publishes the result.</summary>
<description>
Also runs after an unexpected exception interrupts the case.
</description>
*)
METHOD PROTECTED AfterTest
_Stack.Clear();
END_METHOD

//! <summary>Borrows the concrete class name. Callers must not modify it.</summary>
{attribute 'monitoring' := 'call'}
PROPERTY ClassName : REFERENCE TO STRING
GET
ClassName REF= _ClassName;
END_GET
END_PROPERTY

//! <summary>Borrows the compiler-initialized namespace name. Callers must not modify it.</summary>
{attribute 'monitoring' := 'call'}
PROPERTY NamespaceName : REFERENCE TO STRING
GET
NamespaceName REF= CurrentNamespace.Name;
END_GET
END_PROPERTY

//! <summary>Reports the concrete instance size in bytes.</summary>
{attribute 'monitoring' := 'call'}
PROPERTY SelfSize : ULINT
GET
SelfSize := XSIZEOF(THIS^);
END_GET
END_PROPERTY

END_FUNCTION_BLOCK

// ---- Tests/Collections/StackRemoveLastTest.TcPOU
(*
SPDX-FileCopyrightText: c 2026 Oleksandr Tiutyk <trofimich@gmail.com>
SPDX-License-Identifier: MIT
License: https://opensource.org/license/mit
*)

(*!
<summary>Checks LIFO removal through empty and reuse of retained storage.</summary>
<description>
Borrows a group-owned stack reserved for this case. Use from one task at a stable address.
Teardown clears the stack and test-owned resources before publication.
</description>
*)

{attribute 'no_assign'}
{attribute 'no_explicit_call' := 'do not call this function block directly'}
FUNCTION_BLOCK StackRemoveLastTest EXTENDS TOF_Testing.SingleCycleTest
VAR_STAT
	{attribute 'hide'}
	_ClassName : STRING := __POUNAME();
END_VAR
VAR
	_Stack : TOF_Collections.IStack;
END_VAR

(*!
<summary>Clears the fixture before the runner publishes the result.</summary>
<description>
Also runs after an unexpected exception interrupts the case.
</description>
*)
METHOD PROTECTED AfterTest
_Stack.Clear();
END_METHOD

//! <summary>Borrows the concrete class name. Callers must not modify it.</summary>
{attribute 'monitoring' := 'call'}
PROPERTY ClassName : REFERENCE TO STRING
GET
ClassName REF= _ClassName;
END_GET
END_PROPERTY

(*!
<summary>Checks LIFO removal through empty and reuse of retained storage.</summary>
*)
METHOD PROTECTED ExecuteTest
VAR
	values : ARRAY [1..4] OF INT := [11, 22, 33, 44];
	usedCapacity : DINT;
END_VAR
_Stack.PushCopy(value := values[1]);
_Stack.PushCopy(value := values[2]);
_Stack.PushCopy(value := values[3]);

usedCapacity := _Stack.Capacity;

_Stack.RemoveLast();

Assert.ThatInt(
	actual := _Stack.Peek().AsInt(),
	message := "Removing the top must reveal the second entry"
).ToBe(expected := values[2]);

Assert.ThatDInt(
	actual := _Stack.Length,
	message := "Removing one entry must leave two"
).ToBe(expected := DINT#2);

_Stack.RemoveLast();

Assert.ThatInt(
	actual := _Stack.Peek().AsInt(),
	message := "Removing the next top must reveal the first entry"
).ToBe(expected := values[1]);

_Stack.RemoveLast();

Assert.ThatBool(
	actual := _Stack.Empty AND_THEN _Stack.Capacity = usedCapacity,
	message := "Removing the last entry must leave empty storage available for reuse"
).IsTrue();

_Stack.PushCopy(value := values[4]);

Assert.ThatInt(
	actual := _Stack.Peek().AsInt(),
	message := "Push after draining must expose the new top"
).ToBe(expected := values[4]);
END_METHOD

(*!
<summary>Binds the stack fixture for this case.</summary>
<description>
Stores a borrowed interface without invoking the fixture. The owning group keeps it alive and
reserves it for this case. TestElement initializes the name and parent.
</description>
<param name="name">Display name of this case.</param>
<param name="parent">Group that owns this case.</param>
<param name="stack">Required live stack reserved for this case.</param>
*)
METHOD FB_init : BOOL
VAR_INPUT
	bInitRetains: BOOL; // TRUE: the retain variables are initialized (reset warm / reset cold)
	bInCopyCode: BOOL; // TRUE: the instance will be copied to the copy code afterward (online change)
	name : WSTRING;
	parent : TOF_Testing.ITestElement;
	stack : TOF_Collections.IStack;
END_VAR
_Stack := stack;
FB_init := TRUE;
END_METHOD

//! <summary>Borrows the compiler-initialized namespace name. Callers must not modify it.</summary>
{attribute 'monitoring' := 'call'}
PROPERTY NamespaceName : REFERENCE TO STRING
GET
NamespaceName REF= CurrentNamespace.Name;
END_GET
END_PROPERTY

//! <summary>Reports the concrete instance size in bytes.</summary>
{attribute 'monitoring' := 'call'}
PROPERTY SelfSize : ULINT
GET
SelfSize := XSIZEOF(THIS^);
END_GET
END_PROPERTY

END_FUNCTION_BLOCK

// ---- Tests/Collections/Static/StaticStackTestGroup.TcPOU
(*
SPDX-FileCopyrightText: c 2026 Oleksandr Tiutyk <trofimich@gmail.com>
SPDX-License-Identifier: MIT
License: https://opensource.org/license/mit
*)

(*!
<summary>Groups fixed-capacity stack storage, LIFO order, cursors, ownership and overflow cases.</summary>
<description>
Owns the cases, their fixed registration array and any fixtures borrowed by the cases.
Each borrowed fixture is reserved for its case throughout the group lifetime. Use from one task at a stable address.
</description>
*)

{attribute 'no_assign'}
{attribute 'no_explicit_call' := 'do not call this function block directly'}
FUNCTION_BLOCK StaticStackTestGroup EXTENDS TOF_Testing.TestGroup<11>
VAR_STAT
	{attribute 'hide'}
	_ClassName : STRING := __POUNAME();
END_VAR
VAR
	_Validator : TOF_Core.GenericValueTypeValidator(typeClass := TOF_Core.GENERIC_TYPE_CLASS.INT_16);
	_OwnedObjectCleanupStack : TOF_Collections.Stack<3>(valueValidator := 0);
	_ValidatorRejectionStack : TOF_Collections.Stack<3>(valueValidator := _Validator);
	_IndexedAccessAndEnumerationStack : TOF_Collections.Stack<3>(valueValidator := 0);
	_EmptyAndIndexBoundsStack : TOF_Collections.Stack<3>(valueValidator := 0);
	_CopiedAndBorrowedValuesStack : TOF_Collections.Stack<3>(valueValidator := 0);
	_ContainsStack : TOF_Collections.Stack<3>(valueValidator := 0);
	_ContainsGenericStack : TOF_Collections.Stack<3>(valueValidator := 0);
	_PushAndPeekStack : TOF_Collections.Stack<3>(valueValidator := 0);
	_RemoveLastStack : TOF_Collections.Stack<3>(valueValidator := 0);

	_OwnedObjectCleanup : StackOwnedObjectCleanupTest(
		name := "OwnedObjectCleanup",
		parent := THIS^,
		stack := _OwnedObjectCleanupStack
	);
	_ValidatorRejection : StackValidatorRejectionTest(
		name := "ValidatorRejection",
		parent := THIS^,
		stack := _ValidatorRejectionStack
	);
	_IndexedAccessAndEnumeration : StackIndexedAccessAndEnumerationTest(
		name := "IndexedAccessAndEnumeration",
		parent := THIS^,
		stack := _IndexedAccessAndEnumerationStack
	);
	_EmptyAndIndexBounds : StackEmptyAndIndexBoundsTest(
		name := "EmptyAndIndexBounds",
		parent := THIS^,
		stack := _EmptyAndIndexBoundsStack
	);
	_CopiedAndBorrowedValues : StackCopiedAndBorrowedValuesTest(
		name := "CopiedAndBorrowedValues",
		parent := THIS^,
		stack := _CopiedAndBorrowedValuesStack
	);
	_Contains : StackContainsTest(name := "Contains", parent := THIS^, stack := _ContainsStack);
	_ContainsGeneric : StackContainsGenericTest(
		name := "ContainsGeneric",
		parent := THIS^,
		stack := _ContainsGenericStack
	);
	_PushAndPeek : StackPushAndPeekTest(name := "PushAndPeek", parent := THIS^, stack := _PushAndPeekStack);
	_Clear : StaticStackClearTest(name := "Clear", parent := THIS^);
	_RemoveLast : StackRemoveLastTest(name := "RemoveLast", parent := THIS^, stack := _RemoveLastStack);
	_Overflow : StaticStackOverflowTest(name := "Overflow", parent := THIS^);

	_Children : ARRAY [0.._ChildCount - 1] OF TOF_Testing.ITestElement :=
	[
		_OwnedObjectCleanup,
		_ValidatorRejection,
		_IndexedAccessAndEnumeration,
		_EmptyAndIndexBounds,
		_CopiedAndBorrowedValues,
		_Contains,
		_ContainsGeneric,
		_PushAndPeek,
		_Clear,
		_RemoveLast,
		_Overflow
	];
END_VAR

//! <summary>Borrows the fixed child array. Callers must not modify it.</summary>
{attribute 'monitoring' := 'call'}
PROPERTY Children : REFERENCE TO ARRAY [0.._ChildCount - 1] OF TOF_Testing.ITestElement
GET
Children REF= _Children;
END_GET
END_PROPERTY

//! <summary>Borrows the concrete class name. Callers must not modify it.</summary>
{attribute 'monitoring' := 'call'}
PROPERTY ClassName : REFERENCE TO STRING
GET
ClassName REF= _ClassName;
END_GET
END_PROPERTY

//! <summary>Borrows the compiler-initialized namespace name. Callers must not modify it.</summary>
{attribute 'monitoring' := 'call'}
PROPERTY NamespaceName : REFERENCE TO STRING
GET
NamespaceName REF= CurrentNamespace.Name;
END_GET
END_PROPERTY

//! <summary>Reports the concrete instance size in bytes.</summary>
{attribute 'monitoring' := 'call'}
PROPERTY SelfSize : ULINT
GET
SelfSize := XSIZEOF(THIS^);
END_GET
END_PROPERTY

END_FUNCTION_BLOCK

// ---- Tests/Collections/Static/StaticStackClearTest.TcPOU
(*
SPDX-FileCopyrightText: c 2026 Oleksandr Tiutyk <trofimich@gmail.com>
SPDX-License-Identifier: MIT
License: https://opensource.org/license/mit
*)

(*!
<summary>Checks populated clear, storage policy and reuse.</summary>
<description>
Owns a stack and its copied values at a stable address. Use from one task.
Teardown clears surviving entries before publication.
</description>
*)

{attribute 'no_assign'}
{attribute 'no_explicit_call' := 'do not call this function block directly'}
FUNCTION_BLOCK StaticStackClearTest EXTENDS TOF_Testing.SingleCycleTest
VAR_STAT
	{attribute 'hide'}
	_ClassName : STRING := __POUNAME();
END_VAR
VAR
	_Stack : TOF_Collections.Stack<3>(valueValidator := 0);
END_VAR

(*!
<summary>Checks populated clear, storage policy and reuse.</summary>
*)
METHOD PROTECTED ExecuteTest
VAR
	values : ARRAY [1..4] OF INT := [11, 22, 33, 44];
END_VAR
_Stack.PushCopy(value := values[1]);
_Stack.PushCopy(value := values[2]);
_Stack.PushCopy(value := values[3]);

Assert.ThatDInt(
	actual := _Stack.Length,
	message := "Clear fixture must start with three entries"
).ToBe(expected := DINT#3);

_Stack.Clear();

Assert.ThatBool(
	actual := _Stack.Empty AND_THEN _Stack.Length = 0,
	message := "Clear must empty the stack"
).IsTrue();

Assert.ThatDInt(
	actual := _Stack.Capacity,
	message := "Clear must restore the expected storage capacity"
).ToBe(expected := DINT#3);

_Stack.Clear();
_Stack.PushCopy(value := values[4]);

Assert.ThatInt(
	actual := _Stack.Peek().AsInt(),
	message := "The cleared stack must expose the fresh top"
).ToBe(expected := values[4]);

Assert.ThatDInt(
	actual := _Stack.Length,
	message := "Reuse must leave only one entry"
).ToBe(expected := DINT#1);
END_METHOD

(*!
<summary>Clears the fixture before the runner publishes the result.</summary>
<description>
Also runs after an unexpected exception interrupts the case.
</description>
*)
METHOD PROTECTED AfterTest
_Stack.Clear();
END_METHOD

//! <summary>Borrows the concrete class name. Callers must not modify it.</summary>
{attribute 'monitoring' := 'call'}
PROPERTY ClassName : REFERENCE TO STRING
GET
ClassName REF= _ClassName;
END_GET
END_PROPERTY

//! <summary>Borrows the compiler-initialized namespace name. Callers must not modify it.</summary>
{attribute 'monitoring' := 'call'}
PROPERTY NamespaceName : REFERENCE TO STRING
GET
NamespaceName REF= CurrentNamespace.Name;
END_GET
END_PROPERTY

//! <summary>Reports the concrete instance size in bytes.</summary>
{attribute 'monitoring' := 'call'}
PROPERTY SelfSize : ULINT
GET
SelfSize := XSIZEOF(THIS^);
END_GET
END_PROPERTY

END_FUNCTION_BLOCK

// ---- Tests/Collections/Static/StaticStackOverflowTest.TcPOU
(*
SPDX-FileCopyrightText: c 2026 Oleksandr Tiutyk <trofimich@gmail.com>
SPDX-License-Identifier: MIT
License: https://opensource.org/license/mit
*)

(*!
<summary>Checks overflow at three entries and reuse after removing the top.</summary>
<description>
Owns a stack and its copied values at a stable address. Use from one task.
Teardown clears surviving entries before publication.
</description>
*)

{attribute 'no_assign'}
{attribute 'no_explicit_call' := 'do not call this function block directly'}
FUNCTION_BLOCK StaticStackOverflowTest EXTENDS TOF_Testing.SingleCycleTest
VAR_STAT
	{attribute 'hide'}
	_ClassName : STRING := __POUNAME();
END_VAR
VAR
	_Stack : TOF_Collections.Stack<3>(valueValidator := 0);
END_VAR

(*!
<summary>Checks overflow at three entries and reuse after removing the top.</summary>
*)
METHOD PROTECTED ExecuteTest
VAR
	values : ARRAY [1..4] OF INT := [11, 22, 33, 44];
	i : DINT;

	exceptionCode : __SYSTEM.ExceptionCode;
	caught : TOF_Core.IException;
	fullException : TOF_Core.IStaticCollectionFullException;
END_VAR
_Stack.PushCopy(value := values[1]);
_Stack.PushCopy(value := values[2]);
_Stack.PushCopy(value := values[3]);

Assert.ThatBool(
	actual := _Stack.Full,
	message := "Overflow fixture must start full"
).IsTrue();

__TRY
	_Stack.PushCopy(value := values[4]);
__CATCH(exceptionCode)
	caught := TOF_Core.ExceptionManager.GetLastException(
		exceptionCode := exceptionCode,
		catchPointNamespaceName := NamespaceName,
		catchPointPOUName := __POUNAME(),
		catchPointPosition := __POSITION()
	);
__ENDTRY

Assert.ThatBool(
	actual := __QUERYINTERFACE(caught, fullException),
	message := "Pushing beyond capacity must raise StaticCollectionFullException"
).IsTrue();

Assert.ThatBool(
	actual := _Stack.Full AND_THEN _Stack.Length = 3 AND_THEN _Stack.Capacity = 3,
	message := "Rejected push must preserve full length and capacity"
).IsTrue();

FOR i := 0 TO 2 DO
	Assert.ThatInt(
		actual := _Stack.GetByIndex(index := i).AsInt(),
		message := "Rejected push must preserve every entry in top-first order"
	).ToBe(expected := values[3 - i]);
END_FOR

_Stack.RemoveLast();
_Stack.PushCopy(value := values[4]);

Assert.ThatBool(
	actual := _Stack.Full AND_THEN _Stack.Length = 3,
	message := "Pushing after removal must reuse the freed slot"
).IsTrue();

Assert.ThatInt(
	actual := _Stack.Peek().AsInt(),
	message := "Reusing the slot must expose the new top"
).ToBe(expected := values[4]);

Assert.ThatInt(
	actual := _Stack.GetByIndex(index := 1).AsInt(),
	message := "Reusing the slot must preserve the prior entries"
).ToBe(expected := values[2]);
END_METHOD

(*!
<summary>Clears the fixture before the runner publishes the result.</summary>
<description>
Also runs after an unexpected exception interrupts the case.
</description>
*)
METHOD PROTECTED AfterTest
_Stack.Clear();
END_METHOD

//! <summary>Borrows the concrete class name. Callers must not modify it.</summary>
{attribute 'monitoring' := 'call'}
PROPERTY ClassName : REFERENCE TO STRING
GET
ClassName REF= _ClassName;
END_GET
END_PROPERTY

//! <summary>Borrows the compiler-initialized namespace name. Callers must not modify it.</summary>
{attribute 'monitoring' := 'call'}
PROPERTY NamespaceName : REFERENCE TO STRING
GET
NamespaceName REF= CurrentNamespace.Name;
END_GET
END_PROPERTY

//! <summary>Reports the concrete instance size in bytes.</summary>
{attribute 'monitoring' := 'call'}
PROPERTY SelfSize : ULINT
GET
SelfSize := XSIZEOF(THIS^);
END_GET
END_PROPERTY

END_FUNCTION_BLOCK

// ---- Tests/Devices/IO/DevicesIOTestGroup.TcPOU
(*
SPDX-FileCopyrightText: c 2026 Oleksandr Tiutyk <trofimich@gmail.com>
SPDX-License-Identifier: MIT
License: https://opensource.org/license/mit
*)

(*!
<summary>Groups digital and analog device, simulated channel and conversion cases.</summary>
<description>
Owns the independent child instances and their fixed registration array. Use from one PLC task at a stable address.
</description>
*)

{attribute 'no_assign'}
{attribute 'no_explicit_call' := 'do not call this function block directly'}
FUNCTION_BLOCK DevicesIOTestGroup EXTENDS TOF_Testing.TestGroup<17>
VAR_STAT
	{attribute 'hide'}
	_ClassName : STRING := __POUNAME();
END_VAR
VAR
	_TestDigitalInputNormallyOpen : DigitalInputNormallyOpenTest(name := "TestDigitalInputNormallyOpen", parent := THIS^);
	_TestDigitalInputNormallyClosed : DigitalInputNormallyClosedTest(
		name := "TestDigitalInputNormallyClosed",
		parent := THIS^
	);
	_TestDigitalInputUnbound : DigitalInputUnboundTest(name := "TestDigitalInputUnbound", parent := THIS^);
	_TestDigitalOutputNormallyOpen : DigitalOutputNormallyOpenTest(
		name := "TestDigitalOutputNormallyOpen",
		parent := THIS^
	);
	_TestDigitalOutputNormallyClosed : DigitalOutputNormallyClosedTest(
		name := "TestDigitalOutputNormallyClosed",
		parent := THIS^
	);
	_TestDirectAnalogValueConverter : DirectAnalogValueConverterTest(
		name := "TestDirectAnalogValueConverter",
		parent := THIS^
	);
	_TestAnalogInputScalingAndScalarBinding : AnalogInputScalingAndScalarBindingTest(
		name := "TestAnalogInputScalingAndScalarBinding",
		parent := THIS^
	);
	_TestAnalogInputChannelStatusAndErrorReporting : AnalogInputChannelStatusAndErrorReportingTest(
		name := "TestAnalogInputChannelStatusAndErrorReporting",
		parent := THIS^
	);
	_TestAnalogInputConverterRecovery : AnalogInputConverterRecoveryTest(
		name := "TestAnalogInputConverterRecovery",
		parent := THIS^
	);
	_TestAnalogInputCriticalConversionError : AnalogInputCriticalConversionErrorTest(
		name := "TestAnalogInputCriticalConversionError",
		parent := THIS^
	);
	_TestAnalogInputStatusWordIsolation : AnalogInputStatusWordIsolationTest(
		name := "TestAnalogInputStatusWordIsolation",
		parent := THIS^
	);
	_TestAnalogInputStatusBitDecoding : AnalogInputStatusBitDecodingTest(
		name := "TestAnalogInputStatusBitDecoding",
		parent := THIS^
	);
	_TestAnalogOutputScaling : AnalogOutputScalingTest(name := "TestAnalogOutputScaling", parent := THIS^);
	_TestAnalogOutputEqualRawLimits : AnalogOutputEqualRawLimitsTest(
		name := "TestAnalogOutputEqualRawLimits",
		parent := THIS^
	);
	_TestDynamicRangeAnalogValueConverter : DynamicRangeAnalogValueConverterTest(
		name := "TestDynamicRangeAnalogValueConverter",
		parent := THIS^
	);
	_TestStaticConverterCopiesLimits : StaticConverterCopiesLimitsTest(
		name := "TestStaticConverterCopiesLimits",
		parent := THIS^
	);
	_TestRangeConverterBoundaryClampingAndZeroDivision : RangeConverterBoundaryClampingAndZeroDivisionTest(
		name := "TestRangeConverterBoundaryClampingAndZeroDivision",
		parent := THIS^
	);

	_Children : ARRAY [0.._ChildCount - 1] OF TOF_Testing.ITestElement :=
	[
		_TestDigitalInputNormallyOpen,
		_TestDigitalInputNormallyClosed,
		_TestDigitalInputUnbound,
		_TestDigitalOutputNormallyOpen,
		_TestDigitalOutputNormallyClosed,
		_TestDirectAnalogValueConverter,
		_TestAnalogInputScalingAndScalarBinding,
		_TestAnalogInputChannelStatusAndErrorReporting,
		_TestAnalogInputConverterRecovery,
		_TestAnalogInputCriticalConversionError,
		_TestAnalogInputStatusWordIsolation,
		_TestAnalogInputStatusBitDecoding,
		_TestAnalogOutputScaling,
		_TestAnalogOutputEqualRawLimits,
		_TestDynamicRangeAnalogValueConverter,
		_TestStaticConverterCopiesLimits,
		_TestRangeConverterBoundaryClampingAndZeroDivision
	];
END_VAR

//! <summary>Borrows the fixed child array. Callers must not modify it.</summary>
{attribute 'monitoring' := 'call'}
PROPERTY Children : REFERENCE TO ARRAY [0.._ChildCount - 1] OF TOF_Testing.ITestElement
GET
Children REF= _Children;
END_GET
END_PROPERTY

//! <summary>Borrows the concrete class name. Callers must not modify it.</summary>
{attribute 'monitoring' := 'call'}
PROPERTY ClassName : REFERENCE TO STRING
GET
ClassName REF= _ClassName;
END_GET
END_PROPERTY

//! <summary>Borrows the compiler-initialized namespace name. Callers must not modify it.</summary>
{attribute 'monitoring' := 'call'}
PROPERTY NamespaceName : REFERENCE TO STRING
GET
NamespaceName REF= CurrentNamespace.Name;
END_GET
END_PROPERTY

//! <summary>Reports the concrete instance size in bytes.</summary>
{attribute 'monitoring' := 'call'}
PROPERTY SelfSize : ULINT
GET
SelfSize := XSIZEOF(THIS^);
END_GET
END_PROPERTY

END_FUNCTION_BLOCK

// ---- Tests/Devices/IO/DigitalInputNormallyOpenTest.TcPOU
(*
SPDX-FileCopyrightText: c 2026 Oleksandr Tiutyk <trofimich@gmail.com>
SPDX-License-Identifier: MIT
License: https://opensource.org/license/mit
*)

(*!
<summary>Checks normal-open input values and transition detection.</summary>
<description>
Uses a live case-owned automation parent and fresh local device fixtures on every run.
The scenario reads and writes ordinary simulated storage within one task cycle.
</description>
*)

{attribute 'no_assign'}
{attribute 'no_explicit_call' := 'do not call this function block directly'}
FUNCTION_BLOCK DigitalInputNormallyOpenTest EXTENDS TOF_Testing.SingleCycleTest
VAR_STAT
	{attribute 'hide'}
	_ClassName : STRING := __POUNAME();
END_VAR
VAR
	//! <summary>Live parent borrowed by the method-local simulated device.</summary>
	_AutomationRoot : MockAutomationController(name := "DevicesIORoot");
END_VAR

(*!
<summary>Checks normal-open input values and transition detection.</summary>
*)
METHOD PROTECTED ExecuteTest
VAR
	input : TOF_Devices_IO.DigitalInput(name := "DI_NO", parent := _AutomationRoot);
	rawInput : BOOL;
END_VAR
input.Initialize();
input.BindToIO(rawValue := rawInput);

Assert.ThatBool(
	actual := input.BoundToIO,
	message := "DigitalInput should be bound to IO"
).IsTrue();

rawInput := FALSE;
input.ProcessInput();
Assert.ThatBool(
	actual := input.Value,
	message := "Value should be FALSE"
).IsFalse();

rawInput := TRUE;
input.ProcessInput();
Assert.ThatBool(
	actual := input.Value,
	message := "Value should be TRUE"
).IsTrue();
Assert.ThatBool(
	actual := input.Changed,
	message := "Changed should be TRUE on transition"
).IsTrue();

input.ProcessInput();
Assert.ThatBool(
	actual := input.Changed,
	message := "Changed should be FALSE when state remains same"
).IsFalse();
END_METHOD

//! <summary>Borrows the concrete class name. Callers must not modify it.</summary>
{attribute 'monitoring' := 'call'}
PROPERTY ClassName : REFERENCE TO STRING
GET
ClassName REF= _ClassName;
END_GET
END_PROPERTY

//! <summary>Borrows the compiler-initialized namespace name. Callers must not modify it.</summary>
{attribute 'monitoring' := 'call'}
PROPERTY NamespaceName : REFERENCE TO STRING
GET
NamespaceName REF= CurrentNamespace.Name;
END_GET
END_PROPERTY

//! <summary>Reports the concrete instance size in bytes.</summary>
{attribute 'monitoring' := 'call'}
PROPERTY SelfSize : ULINT
GET
SelfSize := XSIZEOF(THIS^);
END_GET
END_PROPERTY

END_FUNCTION_BLOCK

// ---- Tests/Devices/IO/DigitalInputNormallyClosedTest.TcPOU
(*
SPDX-FileCopyrightText: c 2026 Oleksandr Tiutyk <trofimich@gmail.com>
SPDX-License-Identifier: MIT
License: https://opensource.org/license/mit
*)

(*!
<summary>Checks input inversion for a normally closed contact.</summary>
<description>
Uses a live case-owned automation parent and fresh local device fixtures on every run.
The scenario reads and writes ordinary simulated storage within one task cycle.
</description>
*)

{attribute 'no_assign'}
{attribute 'no_explicit_call' := 'do not call this function block directly'}
FUNCTION_BLOCK DigitalInputNormallyClosedTest EXTENDS TOF_Testing.SingleCycleTest
VAR_STAT
	{attribute 'hide'}
	_ClassName : STRING := __POUNAME();
END_VAR
VAR
	//! <summary>Live parent borrowed by the method-local simulated device.</summary>
	_AutomationRoot : MockAutomationController(name := "DevicesIORoot");
END_VAR

(*!
<summary>Checks input inversion for a normally closed contact.</summary>
*)
METHOD PROTECTED ExecuteTest
VAR
	input : TOF_Devices_IO.DigitalInput(name := "DI_NC", parent := _AutomationRoot);
	rawInput : BOOL;
END_VAR
input.Initialize();
input.ContactType := TOF_Devices_IO.CONTACT_TYPE.NORMALLY_CLOSED;
input.BindToIO(rawValue := rawInput);

rawInput := FALSE;
input.ProcessInput();
Assert.ThatBool(
	actual := input.Value,
	message := "Value should be inverted TRUE for NC contact"
).IsTrue();

rawInput := TRUE;
input.ProcessInput();
Assert.ThatBool(
	actual := input.Value,
	message := "Value should be inverted FALSE for NC contact"
).IsFalse();
END_METHOD

//! <summary>Borrows the concrete class name. Callers must not modify it.</summary>
{attribute 'monitoring' := 'call'}
PROPERTY ClassName : REFERENCE TO STRING
GET
ClassName REF= _ClassName;
END_GET
END_PROPERTY

//! <summary>Borrows the compiler-initialized namespace name. Callers must not modify it.</summary>
{attribute 'monitoring' := 'call'}
PROPERTY NamespaceName : REFERENCE TO STRING
GET
NamespaceName REF= CurrentNamespace.Name;
END_GET
END_PROPERTY

//! <summary>Reports the concrete instance size in bytes.</summary>
{attribute 'monitoring' := 'call'}
PROPERTY SelfSize : ULINT
GET
SelfSize := XSIZEOF(THIS^);
END_GET
END_PROPERTY

END_FUNCTION_BLOCK

// ---- Tests/Devices/IO/DigitalInputUnboundTest.TcPOU
(*
SPDX-FileCopyrightText: c 2026 Oleksandr Tiutyk <trofimich@gmail.com>
SPDX-License-Identifier: MIT
License: https://opensource.org/license/mit
*)

(*!
<summary>Checks the unbound input value and diagnostic state.</summary>
<description>
Uses a live case-owned automation parent and fresh local device fixtures on every run.
The scenario reads and writes ordinary simulated storage within one task cycle.
</description>
*)

{attribute 'no_assign'}
{attribute 'no_explicit_call' := 'do not call this function block directly'}
FUNCTION_BLOCK DigitalInputUnboundTest EXTENDS TOF_Testing.SingleCycleTest
VAR_STAT
	{attribute 'hide'}
	_ClassName : STRING := __POUNAME();
END_VAR
VAR
	//! <summary>Live parent borrowed by the method-local simulated device.</summary>
	_AutomationRoot : MockAutomationController(name := "DevicesIORoot");
END_VAR

(*!
<summary>Checks the unbound input value and diagnostic state.</summary>
*)
METHOD PROTECTED ExecuteTest
VAR
	input : TOF_Devices_IO.DigitalInput(name := "DI_Unbound", parent := _AutomationRoot);
END_VAR
input.Initialize();
Assert.ThatBool(
	actual := input.BoundToIO,
	message := "BoundToIO should be FALSE"
).IsFalse();

input.ProcessInput();
Assert.ThatBool(
	actual := input.Value,
	message := "Value should default to FALSE"
).IsFalse();
Assert.ThatBool(
	actual := input.HasError,
	message := "Unbound input should not report error"
).IsFalse();
END_METHOD

//! <summary>Borrows the concrete class name. Callers must not modify it.</summary>
{attribute 'monitoring' := 'call'}
PROPERTY ClassName : REFERENCE TO STRING
GET
ClassName REF= _ClassName;
END_GET
END_PROPERTY

//! <summary>Borrows the compiler-initialized namespace name. Callers must not modify it.</summary>
{attribute 'monitoring' := 'call'}
PROPERTY NamespaceName : REFERENCE TO STRING
GET
NamespaceName REF= CurrentNamespace.Name;
END_GET
END_PROPERTY

//! <summary>Reports the concrete instance size in bytes.</summary>
{attribute 'monitoring' := 'call'}
PROPERTY SelfSize : ULINT
GET
SelfSize := XSIZEOF(THIS^);
END_GET
END_PROPERTY

END_FUNCTION_BLOCK

// ---- Tests/Devices/IO/DigitalOutputNormallyOpenTest.TcPOU
(*
SPDX-FileCopyrightText: c 2026 Oleksandr Tiutyk <trofimich@gmail.com>
SPDX-License-Identifier: MIT
License: https://opensource.org/license/mit
*)

(*!
<summary>Checks output writes and acknowledgements of both transitions.</summary>
<description>
Uses a live case-owned automation parent and fresh local device fixtures on every run.
The scenario reads and writes ordinary simulated storage within one task cycle.
</description>
*)

{attribute 'no_assign'}
{attribute 'no_explicit_call' := 'do not call this function block directly'}
FUNCTION_BLOCK DigitalOutputNormallyOpenTest EXTENDS TOF_Testing.SingleCycleTest
VAR_STAT
	{attribute 'hide'}
	_ClassName : STRING := __POUNAME();
END_VAR
VAR
	//! <summary>Live parent borrowed by the method-local simulated device.</summary>
	_AutomationRoot : MockAutomationController(name := "DevicesIORoot");
END_VAR

(*!
<summary>Checks output writes and acknowledgements of both transitions.</summary>
*)
METHOD PROTECTED ExecuteTest
VAR
	output : TOF_Devices_IO.DigitalOutput(name := "DO_NO", parent := _AutomationRoot);
	rawOutput : BOOL;
END_VAR
output.Initialize();
output.BindToIO(rawValue := rawOutput);

output.Value := TRUE;
Assert.ThatBool(
	actual := output.Changed,
	message := "Changed must be TRUE before processing a new value"
).IsTrue();
output.ProcessOutput();
Assert.ThatBool(
	actual := rawOutput,
	message := "rawOutput should be TRUE"
).IsTrue();
Assert.ThatBool(
	actual := output.Changed,
	message := "Processing acknowledges the current value"
).IsFalse();

